LIN {X 0,Y 466.618,Z 479.703,A -85,B 0,C 180,E1 -7650.864,E2 -7650.864} C_VEL
LIN {X 0,Y 466.661,Z 478.907,A -85,B 0,C 180,E1 -7651.727,E2 -7651.727} C_VEL
LIN {X 0,Y 466.686,Z 477.632,A -85,B 0,C 180,E1 -7652.59,E2 -7652.59} C_VEL
LIN {X 0,Y 466.717,Z 474.683,A -85,B 0,C 180,E1 -7653.887,E2 -7653.887} C_VEL
LIN {X 0,Y 466.72,Z 471.998,A -85,B 0,C 180,E1 -7654.752,E2 -7654.752} C_VEL
LIN {X 0,Y 466.841,Z 466.754,A -85,B 0,C 180,E1 -7656.05,E2 -7656.05} C_VEL
LIN {X 0,Y 467.052,Z 459.848,A -85,B 0,C 180,E1 -7657.35,E2 -7657.35} C_VEL
LIN {X 0,Y 467.254,Z 452.312,A -85,B 0,C 180,E1 -7658.434,E2 -7658.434} C_VEL
LIN {X 0,Y 467.532,Z 444.89,A -85,B 0,C 180,E1 -7659.301,E2 -7659.301} C_VEL
LIN {X 0,Y 467.855,Z 436.955,A -85,B 0,C 180,E1 -7660.058,E2 -7660.058} C_VEL
LIN {X 0,Y 468.228,Z 427.08,A -85,B 0,C 180,E1 -7660.815,E2 -7660.815} C_VEL
LIN {X 0,Y 468.601,Z 415.545,A -85,B 0,C 180,E1 -7661.464,E2 -7661.464} C_VEL
LIN {X 0,Y 467.661,Z 405.502,A -85,B 0,C 180,E1 -7661.898,E2 -7661.898} C_VEL
LIN {X 0,Y 466.839,Z 397.843,A -85,B 0,C 180,E1 -7662.168,E2 -7662.168} C_VEL
LIN {X 0,Y 467.003,Z 388.045,A -85,B 0,C 180,E1 -7665.603,E2 -7665.603} C_VEL
LIN {X 0,Y 467.199,Z 379.627,A -85,B 0,C 180,E1 -7668.612,E2 -7668.612} C_VEL
LIN {X 0,Y 467.394,Z 371.372,A -85,B 0,C 180,E1 -7671.617,E2 -7671.617} C_VEL
LIN {X 0,Y 467.717,Z 362.707,A -85,B 0,C 180,E1 -7674.882,E2 -7674.882} C_VEL
LIN {X 0,Y 468.042,Z 355.361,A -85,B 0,C 180,E1 -7677.743,E2 -7677.743} C_VEL
LIN {X 0,Y 468.487,Z 348.104,A -85,B 0,C 180,E1 -7680.668,E2 -7680.668} C_VEL
LIN {X 0,Y 468.775,Z 342.812,A -85,B 0,C 180,E1 -7682.905,E2 -7682.905} C_VEL
LIN {X 0,Y 468.213,Z 338.68,A -85,B 0,C 180,E1 -7684.778,E2 -7684.778} C_VEL
LIN {X 0,Y 467.554,Z 335.06,A -85,B 0,C 180,E1 -7686.558,E2 -7686.558} C_VEL
LIN {X 0,Y 467.588,Z 335.057,A -85,B 0,C 180,E1 -7689.145,E2 -7689.145} C_VEL
LIN {X 0,Y 467.593,Z 335.059,A -85,B 0,C 180,E1 -7692.567,E2 -7692.567} C_VEL
LIN {X 0,Y 467.572,Z 335.061,A -85,B 0,C 180,E1 -7695.053,E2 -7695.053} C_VEL
LIN {X 0,Y 467.596,Z 335.055,A -85,B 0,C 180,E1 -7697.44,E2 -7697.44} C_VEL
LIN {X 0,Y 467.565,Z 335.058,A -85,B 0,C 180,E1 -7700.853,E2 -7700.853} C_VEL
LIN {X 0,Y 467.566,Z 335.057,A -85,B 0,C 180,E1 -7704.261,E2 -7704.261} C_VEL
LIN {X 0,Y 467.586,Z 335.055,A -85,B 0,C 180,E1 -7707.321,E2 -7707.321} C_VEL
LIN {X 0,Y 467.575,Z 335.057,A -85,B 0,C 180,E1 -7710.668,E2 -7710.668} C_VEL
LIN {X 0,Y 467.622,Z 335.051,A -85,B 0,C 180,E1 -7713.199,E2 -7713.199} C_VEL
LIN {X 0,Y 467.6,Z 335.055,A -85,B 0,C 180,E1 -7716.468,E2 -7716.468} C_VEL
LIN {X 0,Y 467.629,Z 335.05,A -85,B 0,C 180,E1 -7719.777,E2 -7719.777} C_VEL
LIN {X 0,Y 467.604,Z 335.053,A -85,B 0,C 180,E1 -7722.506,E2 -7722.506} C_VEL
LIN {X 0,Y 467.612,Z 335.051,A -85,B 0,C 180,E1 -7725.196,E2 -7725.196} C_VEL
LIN {X 0,Y 467.663,Z 335.044,A -85,B 0,C 180,E1 -7727.854,E2 -7727.854} C_VEL
LIN {X 0,Y 467.675,Z 335.043,A -85,B 0,C 180,E1 -7731.356,E2 -7731.356} C_VEL
LIN {X 0,Y 467.727,Z 335.037,A -85,B 0,C 180,E1 -7733.962,E2 -7733.962} C_VEL
LIN {X 0,Y 467.856,Z 335.021,A -85,B 0,C 180,E1 -7737.416,E2 -7737.416} C_VEL
LIN {X 0,Y 467.887,Z 335.019,A -85,B 0,C 180,E1 -7739.999,E2 -7739.999} C_VEL
LIN {X 0,Y 467.862,Z 335.021,A -85,B 0,C 180,E1 -7742.582,E2 -7742.582} C_VEL
LIN {X 0,Y 467.741,Z 335.037,A -85,B 0,C 180,E1 -7746.036,E2 -7746.036} C_VEL
LIN {X 0,Y 467.673,Z 335.044,A -85,B 0,C 180,E1 -7748.642,E2 -7748.642} C_VEL
LIN {X 0,Y 467.66,Z 335.047,A -85,B 0,C 180,E1 -7752.144,E2 -7752.144} C_VEL
LIN {X 0,Y 467.642,Z 335.051,A -85,B 0,C 180,E1 -7755.694,E2 -7755.694} C_VEL
LIN {X 0,Y 467.417,Z 335.078,A -85,B 0,C 180,E1 -7758.69,E2 -7758.69} C_VEL
LIN {X 0,Y 467.29,Z 335.094,A -85,B 0,C 180,E1 -7759.321,E2 -7759.321} C_VEL
LIN {X 0,Y 467.198,Z 337.07,A -85,B 0,C 180,E1 -7761.162,E2 -7761.162} C_VEL
LIN {X 0,Y 467.108,Z 340.504,A -85,B 0,C 180,E1 -7763.967,E2 -7763.967} C_VEL
LIN {X 0,Y 466.981,Z 344.105,A -85,B 0,C 180,E1 -7766.838,E2 -7766.838} C_VEL
LIN {X 0,Y 466.91,Z 347.81,A -85,B 0,C 180,E1 -7769.782,E2 -7769.782} C_VEL
LIN {X 0,Y 466.826,Z 351.71,A -85,B 0,C 180,E1 -7772.817,E2 -7772.817} C_VEL
LIN {X 0,Y 466.752,Z 355.321,A -85,B 0,C 180,E1 -7775.6,E2 -7775.6} C_VEL
LIN {X 0,Y 466.727,Z 358.475,A -85,B 0,C 180,E1 -7777.969,E2 -7777.969} C_VEL
LIN {X 0,Y 468.58,Z 368.176,A -85,B 0,C 180,E1 -7778.367,E2 -7778.367} C_VEL
LIN {X 0,Y 468.903,Z 373.407,A -85,B 0,C 180,E1 -7778.617,E2 -7778.617} C_VEL
LIN {X 0,Y 468.593,Z 383.394,A -85,B 0,C 180,E1 -7779.181,E2 -7779.181} C_VEL
LIN {X 0,Y 468.295,Z 392.105,A -85,B 0,C 180,E1 -7779.829,E2 -7779.829} C_VEL
LIN {X 0,Y 467.971,Z 400.816,A -85,B 0,C 180,E1 -7780.646,E2 -7780.646} C_VEL
LIN {X 0,Y 467.701,Z 407.331,A -85,B 0,C 180,E1 -7781.388,E2 -7781.388} C_VEL
LIN {X 0,Y 467.497,Z 413.587,A -85,B 0,C 180,E1 -7782.246,E2 -7782.246} C_VEL
LIN {X 0,Y 467.25,Z 419.139,A -85,B 0,C 180,E1 -7783.167,E2 -7783.167} C_VEL
LIN {X 0,Y 467.064,Z 423.734,A -85,B 0,C 180,E1 -7784.093,E2 -7784.093} C_VEL
LIN {X 0,Y 466.925,Z 427.508,A -85,B 0,C 180,E1 -7785.024,E2 -7785.024} C_VEL
LIN {X 0,Y 466.805,Z 431.088,A -85,B 0,C 180,E1 -7786.166,E2 -7786.166} C_VEL
LIN {X 0,Y 466.685,Z 433.719,A -85,B 0,C 180,E1 -7787.337,E2 -7787.337} C_VEL
LIN {X 0,Y 466.627,Z 435.754,A -85,B 0,C 180,E1 -7788.854,E2 -7788.854} C_VEL
LIN {X 0,Y 466.569,Z 436.187,A -85,B 0,C 180,E1 -7790.192,E2 -7790.192} C_VEL
LIN {X 0,Y 466.6,Z 435.02,A -85,B 0,C 180,E1 -7791.862,E2 -7791.862} C_VEL
LIN {X 0,Y 466.741,Z 432.093,A -85,B 0,C 180,E1 -7793.502,E2 -7793.502} C_VEL
LIN {X 0,Y 466.851,Z 428.469,A -85,B 0,C 180,E1 -7794.747,E2 -7794.747} C_VEL
LIN {X 0,Y 467.024,Z 424.162,A -85,B 0,C 180,E1 -7795.857,E2 -7795.857} C_VEL
LIN {X 0,Y 467.161,Z 420.161,A -85,B 0,C 180,E1 -7796.693,E2 -7796.693} C_VEL
LIN {X 0,Y 467.405,Z 414.019,A -85,B 0,C 180,E1 -7797.737,E2 -7797.737} C_VEL
LIN {X 0,Y 467.69,Z 407.605,A -85,B 0,C 180,E1 -7798.625,E2 -7798.625} C_VEL
LIN {X 0,Y 467.927,Z 399.54,A -85,B 0,C 180,E1 -7799.541,E2 -7799.541} C_VEL
LIN {X 0,Y 468.297,Z 389.393,A -85,B 0,C 180,E1 -7800.442,E2 -7800.442} C_VEL
LIN {X 0,Y 468.624,Z 380.078,A -85,B 0,C 180,E1 -7801.075,E2 -7801.075} C_VEL
LIN {X 0,Y 468.822,Z 371.827,A -85,B 0,C 180,E1 -7801.516,E2 -7801.516} C_VEL
LIN {X 0,Y 468.245,Z 366.243,A -85,B 0,C 180,E1 -7801.783,E2 -7801.783} C_VEL
LIN {X 0,Y 466.751,Z 357.961,A -85,B 0,C 180,E1 -7802.113,E2 -7802.113} C_VEL
LIN {X 0,Y 466.785,Z 354.038,A -85,B 0,C 180,E1 -7805.033,E2 -7805.033} C_VEL
LIN {X 0,Y 466.109,Z 353.155,A -85,B 0,C 180,E1 -7805.745,E2 -7805.745} C_VEL
LIN {X 0,Y 463.245,Z 351.852,A -85,B 0,C 180,E1 -7806.904,E2 -7806.904} C_VEL
LIN {X 0,Y 460.832,Z 350.827,A -85,B 0,C 180,E1 -7807.84,E2 -7807.84} C_VEL
LIN {X 0,Y 459.803,Z 349.971,A -85,B 0,C 180,E1 -7808.561,E2 -7808.561} C_VEL
LIN {X 0,Y 459.721,Z 349.657,A -85,B 0,C 180,E1 -7808.805,E2 -7808.805} C_VEL
LIN {X 0,Y 459.833,Z 346.343,A -85,B 0,C 180,E1 -7811.364,E2 -7811.364} C_VEL
LIN {X 0,Y 459.94,Z 342.592,A -85,B 0,C 180,E1 -7814.287,E2 -7814.287} C_VEL
LIN {X 0,Y 460.076,Z 338.085,A -85,B 0,C 180,E1 -7817.855,E2 -7817.855} C_VEL
LIN {X 0,Y 460.088,Z 336.115,A -85,B 0,C 180,E1 -7819.437,E2 -7819.437} C_VEL
LIN {X 0,Y 460.626,Z 335.921,A -85,B 0,C 180,E1 -7822.618,E2 -7822.618} C_VEL
LIN {X 0,Y 460.685,Z 335.914,A -85,B 0,C 180,E1 -7824.747,E2 -7824.747} C_VEL
LIN {X 0,Y 460.815,Z 335.897,A -85,B 0,C 180,E1 -7827.376,E2 -7827.376} C_VEL
LIN {X 0,Y 460.842,Z 335.895,A -85,B 0,C 180,E1 -7829.999,E2 -7829.999} C_VEL
LIN {X 0,Y 460.816,Z 335.897,A -85,B 0,C 180,E1 -7832.621,E2 -7832.621} C_VEL
LIN {X 0,Y 460.706,Z 335.912,A -85,B 0,C 180,E1 -7836.129,E2 -7836.129} C_VEL
LIN {X 0,Y 460.618,Z 335.921,A -85,B 0,C 180,E1 -7838.775,E2 -7838.775} C_VEL
LIN {X 0,Y 460.621,Z 335.921,A -85,B 0,C 180,E1 -7842.456,E2 -7842.456} C_VEL
LIN {X 0,Y 460.587,Z 335.926,A -85,B 0,C 180,E1 -7845.997,E2 -7845.997} C_VEL
LIN {X 0,Y 460.558,Z 335.929,A -85,B 0,C 180,E1 -7848.901,E2 -7848.901} C_VEL
LIN {X 0,Y 460.502,Z 335.939,A -85,B 0,C 180,E1 -7851.485,E2 -7851.485} C_VEL
LIN {X 0,Y 460.529,Z 335.931,A -85,B 0,C 180,E1 -7854.332,E2 -7854.332} C_VEL
LIN {X 0,Y 460.57,Z 335.929,A -85,B 0,C 180,E1 -7857.242,E2 -7857.242} C_VEL
LIN {X 0,Y 460.513,Z 335.934,A -85,B 0,C 180,E1 -7860.238,E2 -7860.238} C_VEL
LIN {X 0,Y 460.515,Z 335.936,A -85,B 0,C 180,E1 -7863.324,E2 -7863.324} C_VEL
LIN {X 0,Y 460.466,Z 335.941,A -85,B 0,C 180,E1 -7866.529,E2 -7866.529} C_VEL
LIN {X 0,Y 460.564,Z 335.928,A -85,B 0,C 180,E1 -7869.857,E2 -7869.857} C_VEL
LIN {X 0,Y 460.527,Z 335.934,A -85,B 0,C 180,E1 -7872.904,E2 -7872.904} C_VEL
LIN {X 0,Y 460.508,Z 335.935,A -85,B 0,C 180,E1 -7875.829,E2 -7875.829} C_VEL
LIN {X 0,Y 460.528,Z 335.934,A -85,B 0,C 180,E1 -7878.99,E2 -7878.99} C_VEL
LIN {X 0,Y 460.533,Z 335.933,A -85,B 0,C 180,E1 -7881.269,E2 -7881.269} C_VEL
LIN {X 0,Y 460.499,Z 335.938,A -85,B 0,C 180,E1 -7884.555,E2 -7884.555} C_VEL
LIN {X 0,Y 460.518,Z 335.934,A -85,B 0,C 180,E1 -7887.716,E2 -7887.716} C_VEL
LIN {X 0,Y 460.533,Z 335.933,A -85,B 0,C 180,E1 -7890.77,E2 -7890.77} C_VEL
LIN {X 0,Y 460.549,Z 335.93,A -85,B 0,C 180,E1 -7893.735,E2 -7893.735} C_VEL
LIN {X 0,Y 460.534,Z 335.934,A -85,B 0,C 180,E1 -7896.625,E2 -7896.625} C_VEL
LIN {X 0,Y 460.559,Z 335.927,A -85,B 0,C 180,E1 -7899.454,E2 -7899.454} C_VEL
LIN {X 0,Y 460.546,Z 335.932,A -85,B 0,C 180,E1 -7902.231,E2 -7902.231} C_VEL
LIN {X 0,Y 460.556,Z 335.929,A -85,B 0,C 180,E1 -7904.966,E2 -7904.966} C_VEL
LIN {X 0,Y 460.616,Z 335.923,A -85,B 0,C 180,E1 -7907.667,E2 -7907.667} C_VEL
LIN {X 0,Y 460.617,Z 335.922,A -85,B 0,C 180,E1 -7911.225,E2 -7911.225} C_VEL
LIN {X 0,Y 460.699,Z 335.913,A -85,B 0,C 180,E1 -7913.871,E2 -7913.871} C_VEL
LIN {X 0,Y 460.815,Z 335.898,A -85,B 0,C 180,E1 -7917.378,E2 -7917.378} C_VEL
LIN {X 0,Y 460.841,Z 335.895,A -85,B 0,C 180,E1 -7920.001,E2 -7920.001} C_VEL
LIN {X 0,Y 460.816,Z 335.897,A -85,B 0,C 180,E1 -7922.623,E2 -7922.623} C_VEL
LIN {X 0,Y 460.699,Z 335.912,A -85,B 0,C 180,E1 -7926.131,E2 -7926.131} C_VEL
LIN {X 0,Y 460.619,Z 335.921,A -85,B 0,C 180,E1 -7928.777,E2 -7928.777} C_VEL
LIN {X 0,Y 460.624,Z 335.921,A -85,B 0,C 180,E1 -7932.458,E2 -7932.458} C_VEL
LIN {X 0,Y 460.59,Z 335.926,A -85,B 0,C 180,E1 -7935.999,E2 -7935.999} C_VEL
LIN {X 0,Y 460.561,Z 335.929,A -85,B 0,C 180,E1 -7938.903,E2 -7938.903} C_VEL
LIN {X 0,Y 460.507,Z 335.937,A -85,B 0,C 180,E1 -7941.487,E2 -7941.487} C_VEL
LIN {X 0,Y 460.534,Z 335.93,A -85,B 0,C 180,E1 -7944.333,E2 -7944.333} C_VEL
LIN {X 0,Y 460.576,Z 335.929,A -85,B 0,C 180,E1 -7947.244,E2 -7947.244} C_VEL
LIN {X 0,Y 460.519,Z 335.933,A -85,B 0,C 180,E1 -7950.24,E2 -7950.24} C_VEL
LIN {X 0,Y 460.522,Z 335.936,A -85,B 0,C 180,E1 -7953.326,E2 -7953.326} C_VEL
LIN {X 0,Y 460.472,Z 335.94,A -85,B 0,C 180,E1 -7956.53,E2 -7956.53} C_VEL
LIN {X 0,Y 460.538,Z 335.933,A -85,B 0,C 180,E1 -7958.899,E2 -7958.899} C_VEL
LIN {X 0,Y 460.517,Z 335.935,A -85,B 0,C 180,E1 -7962.183,E2 -7962.183} C_VEL
LIN {X 0,Y 460.514,Z 335.936,A -85,B 0,C 180,E1 -7965.413,E2 -7965.413} C_VEL
LIN {X 0,Y 460.53,Z 335.934,A -85,B 0,C 180,E1 -7968.398,E2 -7968.398} C_VEL
LIN {X 0,Y 460.522,Z 335.934,A -85,B 0,C 180,E1 -7971.268,E2 -7971.268} C_VEL
LIN {X 0,Y 460.543,Z 336.026,A -85,B 0,C 180,E1 -7973.553,E2 -7973.553} C_VEL
LIN {X 0,Y 461.613,Z 341.991,A -85,B 0,C 180,E1 -7976.242,E2 -7976.242} C_VEL
LIN {X 0,Y 461.711,Z 345.667,A -85,B 0,C 180,E1 -7977.81,E2 -7977.81} C_VEL
LIN {X 0,Y 461.273,Z 353.052,A -85,B 0,C 180,E1 -7980.822,E2 -7980.822} C_VEL
LIN {X 0,Y 460.829,Z 361.444,A -85,B 0,C 180,E1 -7984.132,E2 -7984.132} C_VEL
LIN {X 0,Y 460.494,Z 369.168,A -85,B 0,C 180,E1 -7987.098,E2 -7987.098} C_VEL
LIN {X 0,Y 460.207,Z 377.901,A -85,B 0,C 180,E1 -7990.37,E2 -7990.37} C_VEL
LIN {X 0,Y 460.009,Z 386.643,A -85,B 0,C 180,E1 -7993.583,E2 -7993.583} C_VEL
LIN {X 0,Y 459.783,Z 395.418,A -85,B 0,C 180,E1 -7996.746,E2 -7996.746} C_VEL
LIN {X 0,Y 459.781,Z 398.053,A -85,B 0,C 180,E1 -7997.693,E2 -7997.693} C_VEL
LIN {X 0,Y 461,Z 410.041,A -85,B 0,C 180,E1 -7998.11,E2 -7998.11} C_VEL
LIN {X 0,Y 461.555,Z 417.186,A -85,B 0,C 180,E1 -7998.453,E2 -7998.453} C_VEL
LIN {X 0,Y 461.209,Z 428.346,A -85,B 0,C 180,E1 -7999.132,E2 -7999.132} C_VEL
LIN {X 0,Y 460.876,Z 436.733,A -85,B 0,C 180,E1 -7999.79,E2 -7999.79} C_VEL
LIN {X 0,Y 460.533,Z 444.67,A -85,B 0,C 180,E1 -8000.559,E2 -8000.559} C_VEL
LIN {X 0,Y 460.247,Z 452.093,A -85,B 0,C 180,E1 -8001.439,E2 -8001.439} C_VEL
LIN {X 0,Y 459.972,Z 459.627,A -85,B 0,C 180,E1 -8002.539,E2 -8002.539} C_VEL
LIN {X 0,Y 459.749,Z 466.524,A -85,B 0,C 180,E1 -8003.858,E2 -8003.858} C_VEL
LIN {X 0,Y 459.651,Z 471.744,A -85,B 0,C 180,E1 -8005.177,E2 -8005.177} C_VEL
LIN {X 0,Y 459.611,Z 474.418,A -85,B 0,C 180,E1 -8006.056,E2 -8006.056} C_VEL
LIN {X 0,Y 459.609,Z 477.345,A -85,B 0,C 180,E1 -8007.372,E2 -8007.372} C_VEL
LIN {X 0,Y 459.57,Z 478.608,A -85,B 0,C 180,E1 -8008.248,E2 -8008.248} C_VEL
LIN {X 0,Y 459.551,Z 479.391,A -85,B 0,C 180,E1 -8009.125,E2 -8009.125} C_VEL
LIN {X 0,Y 459.531,Z 479.678,A -85,B 0,C 180,E1 -8010.001,E2 -8010.001} C_VEL
LIN {X 0,Y 459.551,Z 479.371,A -85,B 0,C 180,E1 -8010.877,E2 -8010.877} C_VEL
LIN {X 0,Y 459.57,Z 478.576,A -85,B 0,C 180,E1 -8011.754,E2 -8011.754} C_VEL
LIN {X 0,Y 459.609,Z 477.301,A -85,B 0,C 180,E1 -8012.63,E2 -8012.63} C_VEL
LIN {X 0,Y 459.61,Z 474.35,A -85,B 0,C 180,E1 -8013.947,E2 -8013.947} C_VEL
LIN {X 0,Y 459.651,Z 471.666,A -85,B 0,C 180,E1 -8014.825,E2 -8014.825} C_VEL
LIN {X 0,Y 459.75,Z 466.419,A -85,B 0,C 180,E1 -8016.144,E2 -8016.144} C_VEL
LIN {X 0,Y 459.978,Z 459.518,A -85,B 0,C 180,E1 -8017.463,E2 -8017.463} C_VEL
LIN {X 0,Y 460.218,Z 451.988,A -85,B 0,C 180,E1 -8018.564,E2 -8018.564} C_VEL
LIN {X 0,Y 460.521,Z 444.576,A -85,B 0,C 180,E1 -8019.443,E2 -8019.443} C_VEL
LIN {X 0,Y 460.861,Z 436.653,A -85,B 0,C 180,E1 -8020.212,E2 -8020.212} C_VEL
LIN {X 0,Y 461.176,Z 428.297,A -85,B 0,C 180,E1 -8020.871,E2 -8020.871} C_VEL
LIN {X 0,Y 461.598,Z 417.276,A -85,B 0,C 180,E1 -8021.548,E2 -8021.548} C_VEL
LIN {X 0,Y 460.674,Z 405.859,A -85,B 0,C 180,E1 -8022.064,E2 -8022.064} C_VEL
LIN {X 0,Y 459.735,Z 397.524,A -85,B 0,C 180,E1 -8022.359,E2 -8022.359} C_VEL
LIN {X 0,Y 459.939,Z 388.146,A -85,B 0,C 180,E1 -8025.707,E2 -8025.707} C_VEL
LIN {X 0,Y 460.145,Z 378.789,A -85,B 0,C 180,E1 -8029.125,E2 -8029.125} C_VEL
LIN {X 0,Y 460.356,Z 371.132,A -85,B 0,C 180,E1 -8031.965,E2 -8031.965} C_VEL
LIN {X 0,Y 460.729,Z 362.485,A -85,B 0,C 180,E1 -8035.286,E2 -8035.286} C_VEL
LIN {X 0,Y 461.146,Z 354.024,A -85,B 0,C 180,E1 -8038.691,E2 -8038.691} C_VEL
LIN {X 0,Y 461.544,Z 348.034,A -85,B 0,C 180,E1 -8041.181,E2 -8041.181} C_VEL
LIN {X 0,Y 461.713,Z 343.331,A -85,B 0,C 180,E1 -8043.229,E2 -8043.229} C_VEL
LIN {X 0,Y 461.004,Z 338.695,A -85,B 0,C 180,E1 -8045.403,E2 -8045.403} C_VEL
LIN {X 0,Y 460.519,Z 335.936,A -85,B 0,C 180,E1 -8046.799,E2 -8046.799} C_VEL
LIN {X 0,Y 460.538,Z 335.937,A -85,B 0,C 180,E1 -8049.863,E2 -8049.863} C_VEL
LIN {X 0,Y 460.519,Z 335.941,A -85,B 0,C 180,E1 -8052.901,E2 -8052.901} C_VEL
LIN {X 0,Y 460.513,Z 335.938,A -85,B 0,C 180,E1 -8055.831,E2 -8055.831} C_VEL
LIN {X 0,Y 460.537,Z 335.934,A -85,B 0,C 180,E1 -8058.989,E2 -8058.989} C_VEL
LIN {X 0,Y 460.524,Z 335.936,A -85,B 0,C 180,E1 -8061.266,E2 -8061.266} C_VEL
LIN {X 0,Y 460.515,Z 335.937,A -85,B 0,C 180,E1 -8064.554,E2 -8064.554} C_VEL
LIN {X 0,Y 460.536,Z 335.932,A -85,B 0,C 180,E1 -8067.715,E2 -8067.715} C_VEL
LIN {X 0,Y 460.545,Z 335.932,A -85,B 0,C 180,E1 -8070.769,E2 -8070.769} C_VEL
LIN {X 0,Y 460.566,Z 335.929,A -85,B 0,C 180,E1 -8073.734,E2 -8073.734} C_VEL
LIN {X 0,Y 460.553,Z 335.931,A -85,B 0,C 180,E1 -8076.624,E2 -8076.624} C_VEL
LIN {X 0,Y 460.557,Z 335.929,A -85,B 0,C 180,E1 -8079.452,E2 -8079.452} C_VEL
LIN {X 0,Y 460.556,Z 335.931,A -85,B 0,C 180,E1 -8082.229,E2 -8082.229} C_VEL
LIN {X 0,Y 460.571,Z 335.929,A -85,B 0,C 180,E1 -8084.964,E2 -8084.964} C_VEL
LIN {X 0,Y 460.616,Z 335.923,A -85,B 0,C 180,E1 -8088.559,E2 -8088.559} C_VEL
LIN {X 0,Y 460.625,Z 335.921,A -85,B 0,C 180,E1 -8091.223,E2 -8091.223} C_VEL
LIN {X 0,Y 460.691,Z 335.913,A -85,B 0,C 180,E1 -8093.869,E2 -8093.869} C_VEL
LIN {X 0,Y 460.796,Z 335.901,A -85,B 0,C 180,E1 -8097.377,E2 -8097.377} C_VEL
LIN {X 0,Y 460.857,Z 335.895,A -85,B 0,C 180,E1 -8099.999,E2 -8099.999} C_VEL
LIN {X 0,Y 460.803,Z 335.9,A -85,B 0,C 180,E1 -8102.622,E2 -8102.622} C_VEL
LIN {X 0,Y 460.706,Z 335.913,A -85,B 0,C 180,E1 -8106.129,E2 -8106.129} C_VEL
LIN {X 0,Y 460.623,Z 335.922,A -85,B 0,C 180,E1 -8108.775,E2 -8108.775} C_VEL
LIN {X 0,Y 460.618,Z 335.923,A -85,B 0,C 180,E1 -8112.444,E2 -8112.444} C_VEL
LIN {X 0,Y 460.581,Z 335.93,A -85,B 0,C 180,E1 -8115.987,E2 -8115.987} C_VEL
LIN {X 0,Y 460.34,Z 335.959,A -85,B 0,C 180,E1 -8118.815,E2 -8118.815} C_VEL
LIN {X 0,Y 460.194,Z 336.061,A -85,B 0,C 180,E1 -8119.631,E2 -8119.631} C_VEL
LIN {X 0,Y 460.092,Z 339.461,A -85,B 0,C 180,E1 -8122.449,E2 -8122.449} C_VEL
LIN {X 0,Y 459.98,Z 343.335,A -85,B 0,C 180,E1 -8125.648,E2 -8125.648} C_VEL
LIN {X 0,Y 459.906,Z 346.641,A -85,B 0,C 180,E1 -8128.275,E2 -8128.275} C_VEL
LIN {X 0,Y 459.818,Z 350.456,A -85,B 0,C 180,E1 -8131.308,E2 -8131.308} C_VEL
LIN {X 0,Y 459.724,Z 354.451,A -85,B 0,C 180,E1 -8134.445,E2 -8134.445} C_VEL
LIN {X 0,Y 459.655,Z 358.766,A -85,B 0,C 180,E1 -8137.772,E2 -8137.772} C_VEL
LIN {X 0,Y 461.793,Z 370.032,A -85,B 0,C 180,E1 -8138.258,E2 -8138.258} C_VEL
LIN {X 0,Y 461.881,Z 376.837,A -85,B 0,C 180,E1 -8138.597,E2 -8138.597} C_VEL
LIN {X 0,Y 461.585,Z 385.85,A -85,B 0,C 180,E1 -8139.163,E2 -8139.163} C_VEL
LIN {X 0,Y 461.26,Z 393.763,A -85,B 0,C 180,E1 -8139.785,E2 -8139.785} C_VEL
LIN {X 0,Y 461.016,Z 400.657,A -85,B 0,C 180,E1 -8140.443,E2 -8140.443} C_VEL
LIN {X 0,Y 460.682,Z 408.035,A -85,B 0,C 180,E1 -8141.297,E2 -8141.297} C_VEL
LIN {X 0,Y 460.464,Z 414.342,A -85,B 0,C 180,E1 -8142.186,E2 -8142.186} C_VEL
LIN {X 0,Y 460.11,Z 421.406,A -85,B 0,C 180,E1 -8143.419,E2 -8143.419} C_VEL
LIN {X 0,Y 459.929,Z 426.867,A -85,B 0,C 180,E1 -8144.659,E2 -8144.659} C_VEL
LIN {X 0,Y 459.763,Z 430.963,A -85,B 0,C 180,E1 -8145.925,E2 -8145.925} C_VEL
LIN {X 0,Y 459.611,Z 433.924,A -85,B 0,C 180,E1 -8147.219,E2 -8147.219} C_VEL
LIN {X 0,Y 459.543,Z 435.772,A -85,B 0,C 180,E1 -8148.535,E2 -8148.535} C_VEL
LIN {X 0,Y 459.496,Z 436.55,A -85,B 0,C 180,E1 -8150.029,E2 -8150.029} C_VEL
LIN {X 0,Y 459.485,Z 436.038,A -85,B 0,C 180,E1 -8151.264,E2 -8151.264} C_VEL
LIN {X 0,Y 459.558,Z 434.181,A -85,B 0,C 180,E1 -8152.675,E2 -8152.675} C_VEL
LIN {X 0,Y 459.646,Z 432.817,A -85,B 0,C 180,E1 -8153.393,E2 -8153.393} C_VEL
LIN {X 0,Y 459.757,Z 429.915,A -85,B 0,C 180,E1 -8154.487,E2 -8154.487} C_VEL
LIN {X 0,Y 459.968,Z 424.797,A -85,B 0,C 180,E1 -8155.869,E2 -8155.869} C_VEL
LIN {X 0,Y 460.153,Z 419.781,A -85,B 0,C 180,E1 -8156.921,E2 -8156.921} C_VEL
LIN {X 0,Y 460.326,Z 415.314,A -85,B 0,C 180,E1 -8157.698,E2 -8157.698} C_VEL
LIN {X 0,Y 460.584,Z 409.931,A -85,B 0,C 180,E1 -8158.492,E2 -8158.492} C_VEL
LIN {X 0,Y 460.871,Z 402.393,A -85,B 0,C 180,E1 -8159.405,E2 -8159.405} C_VEL
LIN {X 0,Y 461.116,Z 395.587,A -85,B 0,C 180,E1 -8160.088,E2 -8160.088} C_VEL
LIN {X 0,Y 461.409,Z 387.767,A -85,B 0,C 180,E1 -8160.736,E2 -8160.736} C_VEL
LIN {X 0,Y 461.704,Z 379.555,A -85,B 0,C 180,E1 -8161.285,E2 -8161.285} C_VEL
LIN {X 0,Y 461.898,Z 371.097,A -85,B 0,C 180,E1 -8161.732,E2 -8161.732} C_VEL
LIN {X 0,Y 460.131,Z 360.919,A -85,B 0,C 180,E1 -8162.182,E2 -8162.182} C_VEL
LIN {X 0,Y 459.686,Z 358.242,A -85,B 0,C 180,E1 -8162.308,E2 -8162.308} C_VEL
LIN {X 0,Y 459.695,Z 354.608,A -85,B 0,C 180,E1 -8165.037,E2 -8165.037} C_VEL
LIN {X 0,Y 459.708,Z 351.33,A -85,B 0,C 180,E1 -8167.529,E2 -8167.529} C_VEL
LIN {X 0,Y 459.721,Z 349.657,A -85,B 0,C 180,E1 -8168.805,E2 -8168.805} C_VEL
LIN {X 0,Y 459.063,Z 348.78,A -85,B 0,C 180,E1 -8169.528,E2 -8169.528} C_VEL
LIN {X 0,Y 456.226,Z 347.51,A -85,B 0,C 180,E1 -8170.708,E2 -8170.708} C_VEL
LIN {X 0,Y 453.841,Z 346.514,A -85,B 0,C 180,E1 -8171.66,E2 -8171.66} C_VEL
LIN {X 0,Y 452.842,Z 345.676,A -85,B 0,C 180,E1 -8172.394,E2 -8172.394} C_VEL
LIN {X 0,Y 452.774,Z 345.363,A -85,B 0,C 180,E1 -8172.642,E2 -8172.642} C_VEL
LIN {X 0,Y 452.851,Z 341.597,A -85,B 0,C 180,E1 -8175.621,E2 -8175.621} C_VEL
LIN {X 0,Y 453.018,Z 338.172,A -85,B 0,C 180,E1 -8178.364,E2 -8178.364} C_VEL
LIN {X 0,Y 453.027,Z 337.053,A -85,B 0,C 180,E1 -8179.27,E2 -8179.27} C_VEL
LIN {X 0,Y 453.577,Z 336.8,A -85,B 0,C 180,E1 -8182.581,E2 -8182.581} C_VEL
LIN {X 0,Y 453.657,Z 336.79,A -85,B 0,C 180,E1 -8184.665,E2 -8184.665} C_VEL
LIN {X 0,Y 453.755,Z 336.776,A -85,B 0,C 180,E1 -8187.336,E2 -8187.336} C_VEL
LIN {X 0,Y 453.812,Z 336.771,A -85,B 0,C 180,E1 -8189.999,E2 -8189.999} C_VEL
LIN {X 0,Y 453.756,Z 336.776,A -85,B 0,C 180,E1 -8192.662,E2 -8192.662} C_VEL
LIN {X 0,Y 453.672,Z 336.788,A -85,B 0,C 180,E1 -8196.224,E2 -8196.224} C_VEL
LIN {X 0,Y 453.582,Z 336.797,A -85,B 0,C 180,E1 -8198.912,E2 -8198.912} C_VEL
LIN {X 0,Y 453.589,Z 336.798,A -85,B 0,C 180,E1 -8202.55,E2 -8202.55} C_VEL
LIN {X 0,Y 453.531,Z 336.806,A -85,B 0,C 180,E1 -8206.195,E2 -8206.195} C_VEL
LIN {X 0,Y 453.507,Z 336.808,A -85,B 0,C 180,E1 -8209.04,E2 -8209.04} C_VEL
LIN {X 0,Y 453.463,Z 336.814,A -85,B 0,C 180,E1 -8211.835,E2 -8211.835} C_VEL
LIN {X 0,Y 453.5,Z 336.807,A -85,B 0,C 180,E1 -8214.734,E2 -8214.734} C_VEL
LIN {X 0,Y 453.524,Z 336.805,A -85,B 0,C 180,E1 -8217.961,E2 -8217.961} C_VEL
LIN {X 0,Y 453.469,Z 336.811,A -85,B 0,C 180,E1 -8220.758,E2 -8220.758} C_VEL
LIN {X 0,Y 453.463,Z 336.812,A -85,B 0,C 180,E1 -8223.912,E2 -8223.912} C_VEL
LIN {X 0,Y 453.458,Z 336.816,A -85,B 0,C 180,E1 -8227.187,E2 -8227.187} C_VEL
LIN {X 0,Y 453.518,Z 336.808,A -85,B 0,C 180,E1 -8229.445,E2 -8229.445} C_VEL
LIN {X 0,Y 453.477,Z 336.812,A -85,B 0,C 180,E1 -8232.991,E2 -8232.991} C_VEL
LIN {X 0,Y 453.462,Z 336.813,A -85,B 0,C 180,E1 -8235.78,E2 -8235.78} C_VEL
LIN {X 0,Y 453.481,Z 336.811,A -85,B 0,C 180,E1 -8238.211,E2 -8238.211} C_VEL
LIN {X 0,Y 453.518,Z 336.808,A -85,B 0,C 180,E1 -8240.787,E2 -8240.787} C_VEL
LIN {X 0,Y 453.443,Z 336.814,A -85,B 0,C 180,E1 -8243.918,E2 -8243.918} C_VEL
LIN {X 0,Y 453.468,Z 336.813,A -85,B 0,C 180,E1 -8247.151,E2 -8247.151} C_VEL
LIN {X 0,Y 453.499,Z 336.809,A -85,B 0,C 180,E1 -8250.271,E2 -8250.271} C_VEL
LIN {X 0,Y 453.495,Z 336.808,A -85,B 0,C 180,E1 -8253.295,E2 -8253.295} C_VEL
LIN {X 0,Y 453.492,Z 336.81,A -85,B 0,C 180,E1 -8256.239,E2 -8256.239} C_VEL
LIN {X 0,Y 453.494,Z 336.808,A -85,B 0,C 180,E1 -8259.119,E2 -8259.119} C_VEL
LIN {X 0,Y 453.499,Z 336.809,A -85,B 0,C 180,E1 -8261.945,E2 -8261.945} C_VEL
LIN {X 0,Y 453.536,Z 336.806,A -85,B 0,C 180,E1 -8264.727,E2 -8264.727} C_VEL
LIN {X 0,Y 453.589,Z 336.797,A -85,B 0,C 180,E1 -8267.473,E2 -8267.473} C_VEL
LIN {X 0,Y 453.581,Z 336.798,A -85,B 0,C 180,E1 -8271.087,E2 -8271.087} C_VEL
LIN {X 0,Y 453.666,Z 336.789,A -85,B 0,C 180,E1 -8273.776,E2 -8273.776} C_VEL
LIN {X 0,Y 453.755,Z 336.777,A -85,B 0,C 180,E1 -8277.338,E2 -8277.338} C_VEL
LIN {X 0,Y 453.811,Z 336.771,A -85,B 0,C 180,E1 -8280.001,E2 -8280.001} C_VEL
LIN {X 0,Y 453.757,Z 336.776,A -85,B 0,C 180,E1 -8282.664,E2 -8282.664} C_VEL
LIN {X 0,Y 453.667,Z 336.788,A -85,B 0,C 180,E1 -8286.226,E2 -8286.226} C_VEL
LIN {X 0,Y 453.583,Z 336.797,A -85,B 0,C 180,E1 -8288.914,E2 -8288.914} C_VEL
LIN {X 0,Y 453.591,Z 336.797,A -85,B 0,C 180,E1 -8292.552,E2 -8292.552} C_VEL
LIN {X 0,Y 453.535,Z 336.805,A -85,B 0,C 180,E1 -8296.197,E2 -8296.197} C_VEL
LIN {X 0,Y 453.511,Z 336.808,A -85,B 0,C 180,E1 -8299.042,E2 -8299.042} C_VEL
LIN {X 0,Y 453.467,Z 336.813,A -85,B 0,C 180,E1 -8301.837,E2 -8301.837} C_VEL
LIN {X 0,Y 453.506,Z 336.807,A -85,B 0,C 180,E1 -8304.736,E2 -8304.736} C_VEL
LIN {X 0,Y 453.531,Z 336.804,A -85,B 0,C 180,E1 -8307.962,E2 -8307.962} C_VEL
LIN {X 0,Y 453.475,Z 336.811,A -85,B 0,C 180,E1 -8310.76,E2 -8310.76} C_VEL
LIN {X 0,Y 453.471,Z 336.811,A -85,B 0,C 180,E1 -8313.914,E2 -8313.914} C_VEL
LIN {X 0,Y 453.464,Z 336.815,A -85,B 0,C 180,E1 -8317.189,E2 -8317.189} C_VEL
LIN {X 0,Y 453.499,Z 336.81,A -85,B 0,C 180,E1 -8319.449,E2 -8319.449} C_VEL
LIN {X 0,Y 453.462,Z 336.815,A -85,B 0,C 180,E1 -8322.996,E2 -8322.996} C_VEL
LIN {X 0,Y 453.467,Z 336.812,A -85,B 0,C 180,E1 -8325.781,E2 -8325.781} C_VEL
LIN {X 0,Y 453.476,Z 336.812,A -85,B 0,C 180,E1 -8328.211,E2 -8328.211} C_VEL
LIN {X 0,Y 453.511,Z 336.807,A -85,B 0,C 180,E1 -8330.791,E2 -8330.791} C_VEL
LIN {X 0,Y 453.517,Z 336.992,A -85,B 0,C 180,E1 -8333.403,E2 -8333.403} C_VEL
LIN {X 0,Y 454.596,Z 343.067,A -85,B 0,C 180,E1 -8336.184,E2 -8336.184} C_VEL
LIN {X 0,Y 454.638,Z 347.832,A -85,B 0,C 180,E1 -8338.236,E2 -8338.236} C_VEL
LIN {X 0,Y 454.156,Z 355.343,A -85,B 0,C 180,E1 -8341.334,E2 -8341.334} C_VEL
LIN {X 0,Y 453.752,Z 362.759,A -85,B 0,C 180,E1 -8344.3,E2 -8344.3} C_VEL
LIN {X 0,Y 453.427,Z 370.183,A -85,B 0,C 180,E1 -8347.203,E2 -8347.203} C_VEL
LIN {X 0,Y 453.122,Z 378.885,A -85,B 0,C 180,E1 -8350.522,E2 -8350.522} C_VEL
LIN {X 0,Y 452.898,Z 387.629,A -85,B 0,C 180,E1 -8353.782,E2 -8353.782} C_VEL
LIN {X 0,Y 452.693,Z 396.338,A -85,B 0,C 180,E1 -8356.992,E2 -8356.992} C_VEL
LIN {X 0,Y 452.707,Z 397.739,A -85,B 0,C 180,E1 -8357.505,E2 -8357.505} C_VEL
LIN {X 0,Y 454.03,Z 410.787,A -85,B 0,C 180,E1 -8357.983,E2 -8357.983} C_VEL
LIN {X 0,Y 454.556,Z 418.104,A -85,B 0,C 180,E1 -8358.348,E2 -8358.348} C_VEL
LIN {X 0,Y 454.22,Z 427.901,A -85,B 0,C 180,E1 -8358.962,E2 -8358.962} C_VEL
LIN {X 0,Y 453.852,Z 436.31,A -85,B 0,C 180,E1 -8359.631,E2 -8359.631} C_VEL
LIN {X 0,Y 453.512,Z 444.265,A -85,B 0,C 180,E1 -8360.412,E2 -8360.412} C_VEL
LIN {X 0,Y 453.204,Z 451.704,A -85,B 0,C 180,E1 -8361.305,E2 -8361.305} C_VEL
LIN {X 0,Y 452.899,Z 459.25,A -85,B 0,C 180,E1 -8362.422,E2 -8362.422} C_VEL
LIN {X 0,Y 452.66,Z 466.165,A -85,B 0,C 180,E1 -8363.762,E2 -8363.762} C_VEL
LIN {X 0,Y 452.582,Z 471.394,A -85,B 0,C 180,E1 -8365.102,E2 -8365.102} C_VEL
LIN {X 0,Y 452.509,Z 474.072,A -85,B 0,C 180,E1 -8365.993,E2 -8365.993} C_VEL
LIN {X 0,Y 452.533,Z 477.005,A -85,B 0,C 180,E1 -8367.331,E2 -8367.331} C_VEL
LIN {X 0,Y 452.483,Z 478.27,A -85,B 0,C 180,E1 -8368.221,E2 -8368.221} C_VEL
LIN {X 0,Y 452.486,Z 479.058,A -85,B 0,C 180,E1 -8369.111,E2 -8369.111} C_VEL
LIN {X 0,Y 452.464,Z 479.346,A -85,B 0,C 180,E1 -8370.001,E2 -8370.001} C_VEL
LIN {X 0,Y 452.486,Z 479.04,A -85,B 0,C 180,E1 -8370.891,E2 -8370.891} C_VEL
LIN {X 0,Y 452.483,Z 478.245,A -85,B 0,C 180,E1 -8371.781,E2 -8371.781} C_VEL
LIN {X 0,Y 452.534,Z 476.974,A -85,B 0,C 180,E1 -8372.672,E2 -8372.672} C_VEL
LIN {X 0,Y 452.508,Z 474.024,A -85,B 0,C 180,E1 -8374.009,E2 -8374.009} C_VEL
LIN {X 0,Y 452.582,Z 471.344,A -85,B 0,C 180,E1 -8374.901,E2 -8374.901} C_VEL
LIN {X 0,Y 452.662,Z 466.101,A -85,B 0,C 180,E1 -8376.24,E2 -8376.24} C_VEL
LIN {X 0,Y 452.903,Z 459.207,A -85,B 0,C 180,E1 -8377.58,E2 -8377.58} C_VEL
LIN {X 0,Y 453.188,Z 451.685,A -85,B 0,C 180,E1 -8378.698,E2 -8378.698} C_VEL
LIN {X 0,Y 453.511,Z 444.28,A -85,B 0,C 180,E1 -8379.591,E2 -8379.591} C_VEL
LIN {X 0,Y 453.848,Z 436.365,A -85,B 0,C 180,E1 -8380.372,E2 -8380.372} C_VEL
LIN {X 0,Y 454.202,Z 428.025,A -85,B 0,C 180,E1 -8381.04,E2 -8381.04} C_VEL
LIN {X 0,Y 454.615,Z 417.333,A -85,B 0,C 180,E1 -8381.713,E2 -8381.713} C_VEL
LIN {X 0,Y 453.637,Z 405.688,A -85,B 0,C 180,E1 -8382.254,E2 -8382.254} C_VEL
LIN {X 0,Y 452.666,Z 397.221,A -85,B 0,C 180,E1 -8382.555,E2 -8382.555} C_VEL
LIN {X 0,Y 452.861,Z 388.292,A -85,B 0,C 180,E1 -8385.806,E2 -8385.806} C_VEL
LIN {X 0,Y 453.074,Z 379.663,A -85,B 0,C 180,E1 -8389.012,E2 -8389.012} C_VEL
LIN {X 0,Y 453.307,Z 372.209,A -85,B 0,C 180,E1 -8391.846,E2 -8391.846} C_VEL
LIN {X 0,Y 453.672,Z 363.564,A -85,B 0,C 180,E1 -8395.216,E2 -8395.216} C_VEL
LIN {X 0,Y 454.121,Z 355.112,A -85,B 0,C 180,E1 -8398.671,E2 -8398.671} C_VEL
LIN {X 0,Y 454.528,Z 349.149,A -85,B 0,C 180,E1 -8401.198,E2 -8401.198} C_VEL
LIN {X 0,Y 454.775,Z 345.621,A -85,B 0,C 180,E1 -8402.745,E2 -8402.745} C_VEL
LIN {X 0,Y 454.415,Z 342.145,A -85,B 0,C 180,E1 -8404.362,E2 -8404.362} C_VEL
LIN {X 0,Y 453.479,Z 336.813,A -85,B 0,C 180,E1 -8407.073,E2 -8407.073} C_VEL
LIN {X 0,Y 453.511,Z 336.813,A -85,B 0,C 180,E1 -8409.449,E2 -8409.449} C_VEL
LIN {X 0,Y 453.469,Z 336.819,A -85,B 0,C 180,E1 -8412.995,E2 -8412.995} C_VEL
LIN {X 0,Y 453.468,Z 336.815,A -85,B 0,C 180,E1 -8415.779,E2 -8415.779} C_VEL
LIN {X 0,Y 453.486,Z 336.811,A -85,B 0,C 180,E1 -8418.209,E2 -8418.209} C_VEL
LIN {X 0,Y 453.477,Z 336.812,A -85,B 0,C 180,E1 -8420.797,E2 -8420.797} C_VEL
LIN {X 0,Y 453.46,Z 336.814,A -85,B 0,C 180,E1 -8423.917,E2 -8423.917} C_VEL
LIN {X 0,Y 453.485,Z 336.812,A -85,B 0,C 180,E1 -8427.151,E2 -8427.151} C_VEL
LIN {X 0,Y 453.48,Z 336.812,A -85,B 0,C 180,E1 -8430.268,E2 -8430.268} C_VEL
LIN {X 0,Y 453.511,Z 336.808,A -85,B 0,C 180,E1 -8433.294,E2 -8433.294} C_VEL
LIN {X 0,Y 453.509,Z 336.809,A -85,B 0,C 180,E1 -8436.238,E2 -8436.238} C_VEL
LIN {X 0,Y 453.489,Z 336.811,A -85,B 0,C 180,E1 -8439.117,E2 -8439.117} C_VEL
LIN {X 0,Y 453.51,Z 336.807,A -85,B 0,C 180,E1 -8441.944,E2 -8441.944} C_VEL
LIN {X 0,Y 453.546,Z 336.805,A -85,B 0,C 180,E1 -8444.726,E2 -8444.726} C_VEL
LIN {X 0,Y 453.565,Z 336.802,A -85,B 0,C 180,E1 -8448.378,E2 -8448.378} C_VEL
LIN {X 0,Y 453.591,Z 336.798,A -85,B 0,C 180,E1 -8451.086,E2 -8451.086} C_VEL
LIN {X 0,Y 453.657,Z 336.789,A -85,B 0,C 180,E1 -8453.774,E2 -8453.774} C_VEL
LIN {X 0,Y 453.74,Z 336.779,A -85,B 0,C 180,E1 -8457.336,E2 -8457.336} C_VEL
LIN {X 0,Y 453.828,Z 336.77,A -85,B 0,C 180,E1 -8459.999,E2 -8459.999} C_VEL
LIN {X 0,Y 453.747,Z 336.778,A -85,B 0,C 180,E1 -8462.662,E2 -8462.662} C_VEL
LIN {X 0,Y 453.673,Z 336.789,A -85,B 0,C 180,E1 -8466.224,E2 -8466.224} C_VEL
LIN {X 0,Y 453.589,Z 336.798,A -85,B 0,C 180,E1 -8468.912,E2 -8468.912} C_VEL
LIN {X 0,Y 453.568,Z 336.801,A -85,B 0,C 180,E1 -8472.528,E2 -8472.528} C_VEL
LIN {X 0,Y 453.538,Z 336.808,A -85,B 0,C 180,E1 -8476.195,E2 -8476.195} C_VEL
LIN {X 0,Y 453.27,Z 336.84,A -85,B 0,C 180,E1 -8479.001,E2 -8479.001} C_VEL
LIN {X 0,Y 453.119,Z 337.302,A -85,B 0,C 180,E1 -8479.95,E2 -8479.95} C_VEL
LIN {X 0,Y 453.014,Z 340.712,A -85,B 0,C 180,E1 -8482.819,E2 -8482.819} C_VEL
LIN {X 0,Y 452.901,Z 344.352,A -85,B 0,C 180,E1 -8485.837,E2 -8485.837} C_VEL
LIN {X 0,Y 452.83,Z 347.936,A -85,B 0,C 180,E1 -8488.758,E2 -8488.758} C_VEL
LIN {X 0,Y 452.72,Z 351.815,A -85,B 0,C 180,E1 -8491.856,E2 -8491.856} C_VEL
LIN {X 0,Y 452.619,Z 355.896,A -85,B 0,C 180,E1 -8495.064,E2 -8495.064} C_VEL
LIN {X 0,Y 452.603,Z 359.099,A -85,B 0,C 180,E1 -8497.563,E2 -8497.563} C_VEL
LIN {X 0,Y 454.773,Z 370.57,A -85,B 0,C 180,E1 -8498.076,E2 -8498.076} C_VEL
LIN {X 0,Y 454.962,Z 376.488,A -85,B 0,C 180,E1 -8498.373,E2 -8498.373} C_VEL
LIN {X 0,Y 454.629,Z 386.918,A -85,B 0,C 180,E1 -8499.044,E2 -8499.044} C_VEL
LIN {X 0,Y 454.291,Z 394.442,A -85,B 0,C 180,E1 -8499.652,E2 -8499.652} C_VEL
LIN {X 0,Y 454.004,Z 402.068,A -85,B 0,C 180,E1 -8500.406,E2 -8500.406} C_VEL
LIN {X 0,Y 453.687,Z 408.571,A -85,B 0,C 180,E1 -8501.181,E2 -8501.181} C_VEL
LIN {X 0,Y 453.472,Z 413.897,A -85,B 0,C 180,E1 -8501.933,E2 -8501.933} C_VEL
LIN {X 0,Y 453.153,Z 420.282,A -85,B 0,C 180,E1 -8503.03,E2 -8503.03} C_VEL
LIN {X 0,Y 452.958,Z 424.832,A -85,B 0,C 180,E1 -8503.995,E2 -8503.995} C_VEL
LIN {X 0,Y 452.778,Z 428.809,A -85,B 0,C 180,E1 -8505.042,E2 -8505.042} C_VEL
LIN {X 0,Y 452.732,Z 430.876,A -85,B 0,C 180,E1 -8505.687,E2 -8505.687} C_VEL
LIN {X 0,Y 452.564,Z 433.777,A -85,B 0,C 180,E1 -8506.898,E2 -8506.898} C_VEL
LIN {X 0,Y 452.467,Z 435.792,A -85,B 0,C 180,E1 -8508.206,E2 -8508.206} C_VEL
LIN {X 0,Y 452.393,Z 436.752,A -85,B 0,C 180,E1 -8509.57,E2 -8509.57} C_VEL
LIN {X 0,Y 452.4,Z 436.561,A -85,B 0,C 180,E1 -8510.961,E2 -8510.961} C_VEL
LIN {X 0,Y 452.471,Z 435.096,A -85,B 0,C 180,E1 -8512.385,E2 -8512.385} C_VEL
LIN {X 0,Y 452.595,Z 432.105,A -85,B 0,C 180,E1 -8513.847,E2 -8513.847} C_VEL
LIN {X 0,Y 452.719,Z 428.912,A -85,B 0,C 180,E1 -8514.942,E2 -8514.942} C_VEL
LIN {X 0,Y 452.919,Z 424.75,A -85,B 0,C 180,E1 -8516.039,E2 -8516.039} C_VEL
LIN {X 0,Y 453.12,Z 419.576,A -85,B 0,C 180,E1 -8517.121,E2 -8517.121} C_VEL
LIN {X 0,Y 453.439,Z 413.16,A -85,B 0,C 180,E1 -8518.198,E2 -8518.198} C_VEL
LIN {X 0,Y 453.836,Z 404.213,A -85,B 0,C 180,E1 -8519.377,E2 -8519.377} C_VEL
LIN {X 0,Y 454.096,Z 396.721,A -85,B 0,C 180,E1 -8520.161,E2 -8520.161} C_VEL
LIN {X 0,Y 454.409,Z 388.748,A -85,B 0,C 180,E1 -8520.843,E2 -8520.843} C_VEL
LIN {X 0,Y 454.659,Z 381.282,A -85,B 0,C 180,E1 -8521.366,E2 -8521.366} C_VEL
LIN {X 0,Y 454.933,Z 371.763,A -85,B 0,C 180,E1 -8521.888,E2 -8521.888} C_VEL
LIN {X 0,Y 453.325,Z 362.669,A -85,B 0,C 180,E1 -8522.308,E2 -8522.308} C_VEL
LIN {X 0,Y 452.616,Z 358.553,A -85,B 0,C 180,E1 -8522.486,E2 -8522.486} C_VEL
LIN {X 0,Y 452.61,Z 354.956,A -85,B 0,C 180,E1 -8525.212,E2 -8525.212} C_VEL
LIN {X 0,Y 452.656,Z 350.44,A -85,B 0,C 180,E1 -8528.676,E2 -8528.676} C_VEL
LIN {X 0,Y 452.77,Z 346.297,A -85,B 0,C 180,E1 -8531.913,E2 -8531.913} C_VEL
LIN {X 0,Y 452.774,Z 345.363,A -85,B 0,C 180,E1 -8532.642,E2 -8532.642} C_VEL
LIN {X 0,Y 452.145,Z 344.49,A -85,B 0,C 180,E1 -8533.376,E2 -8533.376} C_VEL
LIN {X 0,Y 449.317,Z 343.26,A -85,B 0,C 180,E1 -8534.573,E2 -8534.573} C_VEL
LIN {X 0,Y 446.916,Z 342.296,A -85,B 0,C 180,E1 -8535.539,E2 -8535.539} C_VEL
LIN {X 0,Y 445.899,Z 341.477,A -85,B 0,C 180,E1 -8536.284,E2 -8536.284} C_VEL
LIN {X 0,Y 445.825,Z 341.169,A -85,B 0,C 180,E1 -8536.535,E2 -8536.535} C_VEL
LIN {X 0,Y 445.973,Z 338.01,A -85,B 0,C 180,E1 -8539.098,E2 -8539.098} C_VEL
LIN {X 0,Y 446.382,Z 337.697,A -85,B 0,C 180,E1 -8541.853,E2 -8541.853} C_VEL
LIN {X 0,Y 446.63,Z 337.666,A -85,B 0,C 180,E1 -8544.581,E2 -8544.581} C_VEL
LIN {X 0,Y 446.699,Z 337.655,A -85,B 0,C 180,E1 -8547.294,E2 -8547.294} C_VEL
LIN {X 0,Y 446.783,Z 337.647,A -85,B 0,C 180,E1 -8549.999,E2 -8549.999} C_VEL
LIN {X 0,Y 446.7,Z 337.655,A -85,B 0,C 180,E1 -8552.704,E2 -8552.704} C_VEL
LIN {X 0,Y 446.641,Z 337.664,A -85,B 0,C 180,E1 -8556.323,E2 -8556.323} C_VEL
LIN {X 0,Y 446.528,Z 337.676,A -85,B 0,C 180,E1 -8559.054,E2 -8559.054} C_VEL
LIN {X 0,Y 446.521,Z 337.677,A -85,B 0,C 180,E1 -8562.728,E2 -8562.728} C_VEL
LIN {X 0,Y 446.477,Z 337.683,A -85,B 0,C 180,E1 -8566.458,E2 -8566.458} C_VEL
LIN {X 0,Y 446.456,Z 337.688,A -85,B 0,C 180,E1 -8569.302,E2 -8569.302} C_VEL
LIN {X 0,Y 446.404,Z 337.693,A -85,B 0,C 180,E1 -8572.199,E2 -8572.199} C_VEL
LIN {X 0,Y 446.444,Z 337.688,A -85,B 0,C 180,E1 -8575.152,E2 -8575.152} C_VEL
LIN {X 0,Y 446.47,Z 337.684,A -85,B 0,C 180,E1 -8578.178,E2 -8578.178} C_VEL
LIN {X 0,Y 446.406,Z 337.695,A -85,B 0,C 180,E1 -8581.299,E2 -8581.299} C_VEL
LIN {X 0,Y 446.416,Z 337.689,A -85,B 0,C 180,E1 -8584.522,E2 -8584.522} C_VEL
LIN {X 0,Y 446.424,Z 337.689,A -85,B 0,C 180,E1 -8588.083,E2 -8588.083} C_VEL
LIN {X 0,Y 446.433,Z 337.691,A -85,B 0,C 180,E1 -8590.921,E2 -8590.921} C_VEL
LIN {X 0,Y 446.43,Z 337.688,A -85,B 0,C 180,E1 -8593.84,E2 -8593.84} C_VEL
LIN {X 0,Y 446.432,Z 337.689,A -85,B 0,C 180,E1 -8596.397,E2 -8596.397} C_VEL
LIN {X 0,Y 446.454,Z 337.684,A -85,B 0,C 180,E1 -8599.805,E2 -8599.805} C_VEL
LIN {X 0,Y 446.42,Z 337.69,A -85,B 0,C 180,E1 -8602.124,E2 -8602.124} C_VEL
LIN {X 0,Y 446.416,Z 337.691,A -85,B 0,C 180,E1 -8605.477,E2 -8605.477} C_VEL
LIN {X 0,Y 446.405,Z 337.693,A -85,B 0,C 180,E1 -8608.7,E2 -8608.7} C_VEL
LIN {X 0,Y 446.47,Z 337.684,A -85,B 0,C 180,E1 -8611.822,E2 -8611.822} C_VEL
LIN {X 0,Y 446.445,Z 337.689,A -85,B 0,C 180,E1 -8614.848,E2 -8614.848} C_VEL
LIN {X 0,Y 446.458,Z 337.686,A -85,B 0,C 180,E1 -8618.238,E2 -8618.238} C_VEL
LIN {X 0,Y 446.444,Z 337.687,A -85,B 0,C 180,E1 -8621.65,E2 -8621.65} C_VEL
LIN {X 0,Y 446.503,Z 337.681,A -85,B 0,C 180,E1 -8624.481,E2 -8624.481} C_VEL
LIN {X 0,Y 446.526,Z 337.678,A -85,B 0,C 180,E1 -8628.194,E2 -8628.194} C_VEL
LIN {X 0,Y 446.588,Z 337.67,A -85,B 0,C 180,E1 -8631.859,E2 -8631.859} C_VEL
LIN {X 0,Y 446.635,Z 337.664,A -85,B 0,C 180,E1 -8634.583,E2 -8634.583} C_VEL
LIN {X 0,Y 446.699,Z 337.656,A -85,B 0,C 180,E1 -8637.296,E2 -8637.296} C_VEL
LIN {X 0,Y 446.782,Z 337.646,A -85,B 0,C 180,E1 -8640.001,E2 -8640.001} C_VEL
LIN {X 0,Y 446.701,Z 337.655,A -85,B 0,C 180,E1 -8642.706,E2 -8642.706} C_VEL
LIN {X 0,Y 446.636,Z 337.664,A -85,B 0,C 180,E1 -8646.325,E2 -8646.325} C_VEL
LIN {X 0,Y 446.529,Z 337.676,A -85,B 0,C 180,E1 -8649.056,E2 -8649.056} C_VEL
LIN {X 0,Y 446.524,Z 337.677,A -85,B 0,C 180,E1 -8652.73,E2 -8652.73} C_VEL
LIN {X 0,Y 446.48,Z 337.682,A -85,B 0,C 180,E1 -8656.46,E2 -8656.46} C_VEL
LIN {X 0,Y 446.46,Z 337.687,A -85,B 0,C 180,E1 -8659.304,E2 -8659.304} C_VEL
LIN {X 0,Y 446.409,Z 337.691,A -85,B 0,C 180,E1 -8662.201,E2 -8662.201} C_VEL
LIN {X 0,Y 446.45,Z 337.689,A -85,B 0,C 180,E1 -8665.153,E2 -8665.153} C_VEL
LIN {X 0,Y 446.476,Z 337.682,A -85,B 0,C 180,E1 -8668.18,E2 -8668.18} C_VEL
LIN {X 0,Y 446.412,Z 337.693,A -85,B 0,C 180,E1 -8671.301,E2 -8671.301} C_VEL
LIN {X 0,Y 446.423,Z 337.689,A -85,B 0,C 180,E1 -8674.524,E2 -8674.524} C_VEL
LIN {X 0,Y 446.424,Z 337.689,A -85,B 0,C 180,E1 -8678.083,E2 -8678.083} C_VEL
LIN {X 0,Y 446.421,Z 337.692,A -85,B 0,C 180,E1 -8680.919,E2 -8680.919} C_VEL
LIN {X 0,Y 446.417,Z 337.689,A -85,B 0,C 180,E1 -8683.845,E2 -8683.845} C_VEL
LIN {X 0,Y 446.415,Z 337.691,A -85,B 0,C 180,E1 -8686.402,E2 -8686.402} C_VEL
LIN {X 0,Y 446.446,Z 337.687,A -85,B 0,C 180,E1 -8689.804,E2 -8689.804} C_VEL
LIN {X 0,Y 446.445,Z 337.69,A -85,B 0,C 180,E1 -8693.12,E2 -8693.12} C_VEL
LIN {X 0,Y 447.399,Z 342.891,A -85,B 0,C 180,E1 -8695.564,E2 -8695.564} C_VEL
LIN {X 0,Y 447.728,Z 346.566,A -85,B 0,C 180,E1 -8697.213,E2 -8697.213} C_VEL
LIN {X 0,Y 447.274,Z 353.922,A -85,B 0,C 180,E1 -8700.335,E2 -8700.335} C_VEL
LIN {X 0,Y 446.784,Z 362.167,A -85,B 0,C 180,E1 -8703.718,E2 -8703.718} C_VEL
LIN {X 0,Y 446.403,Z 369.959,A -85,B 0,C 180,E1 -8706.823,E2 -8706.823} C_VEL
LIN {X 0,Y 446.099,Z 378.632,A -85,B 0,C 180,E1 -8710.203,E2 -8710.203} C_VEL
LIN {X 0,Y 445.844,Z 387.326,A -85,B 0,C 180,E1 -8713.518,E2 -8713.518} C_VEL
LIN {X 0,Y 445.606,Z 396.038,A -85,B 0,C 180,E1 -8716.781,E2 -8716.781} C_VEL
LIN {X 0,Y 445.6,Z 397.451,A -85,B 0,C 180,E1 -8717.308,E2 -8717.308} C_VEL
LIN {X 0,Y 446.942,Z 410.26,A -85,B 0,C 180,E1 -8717.79,E2 -8717.79} C_VEL
LIN {X 0,Y 447.546,Z 418.605,A -85,B 0,C 180,E1 -8718.222,E2 -8718.222} C_VEL
LIN {X 0,Y 447.224,Z 427.449,A -85,B 0,C 180,E1 -8718.788,E2 -8718.788} C_VEL
LIN {X 0,Y 446.832,Z 435.878,A -85,B 0,C 180,E1 -8719.466,E2 -8719.466} C_VEL
LIN {X 0,Y 446.475,Z 443.85,A -85,B 0,C 180,E1 -8720.259,E2 -8720.259} C_VEL
LIN {X 0,Y 446.243,Z 449.592,A -85,B 0,C 180,E1 -8720.94,E2 -8720.94} C_VEL
LIN {X 0,Y 445.955,Z 456.008,A -85,B 0,C 180,E1 -8721.847,E2 -8721.847} C_VEL
LIN {X 0,Y 445.755,Z 461.345,A -85,B 0,C 180,E1 -8722.755,E2 -8722.755} C_VEL
LIN {X 0,Y 445.577,Z 465.796,A -85,B 0,C 180,E1 -8723.662,E2 -8723.662} C_VEL
LIN {X 0,Y 445.513,Z 471.034,A -85,B 0,C 180,E1 -8725.024,E2 -8725.024} C_VEL
LIN {X 0,Y 445.414,Z 473.719,A -85,B 0,C 180,E1 -8725.93,E2 -8725.93} C_VEL
LIN {X 0,Y 445.459,Z 476.659,A -85,B 0,C 180,E1 -8727.288,E2 -8727.288} C_VEL
LIN {X 0,Y 445.399,Z 477.93,A -85,B 0,C 180,E1 -8728.193,E2 -8728.193} C_VEL
LIN {X 0,Y 445.393,Z 478.723,A -85,B 0,C 180,E1 -8729.097,E2 -8729.097} C_VEL
LIN {X 0,Y 445.4,Z 479.013,A -85,B 0,C 180,E1 -8730.001,E2 -8730.001} C_VEL
LIN {X 0,Y 445.393,Z 478.708,A -85,B 0,C 180,E1 -8730.905,E2 -8730.905} C_VEL
LIN {X 0,Y 445.4,Z 477.919,A -85,B 0,C 180,E1 -8731.81,E2 -8731.81} C_VEL
LIN {X 0,Y 445.459,Z 476.65,A -85,B 0,C 180,E1 -8732.714,E2 -8732.714} C_VEL
LIN {X 0,Y 445.413,Z 473.702,A -85,B 0,C 180,E1 -8734.073,E2 -8734.073} C_VEL
LIN {X 0,Y 445.514,Z 471.026,A -85,B 0,C 180,E1 -8734.979,E2 -8734.979} C_VEL
LIN {X 0,Y 445.579,Z 465.783,A -85,B 0,C 180,E1 -8736.34,E2 -8736.34} C_VEL
LIN {X 0,Y 445.855,Z 458.898,A -85,B 0,C 180,E1 -8737.701,E2 -8737.701} C_VEL
LIN {X 0,Y 446.141,Z 451.381,A -85,B 0,C 180,E1 -8738.836,E2 -8738.836} C_VEL
LIN {X 0,Y 446.487,Z 443.982,A -85,B 0,C 180,E1 -8739.743,E2 -8739.743} C_VEL
LIN {X 0,Y 446.84,Z 436.077,A -85,B 0,C 180,E1 -8740.536,E2 -8740.536} C_VEL
LIN {X 0,Y 447.235,Z 427.752,A -85,B 0,C 180,E1 -8741.215,E2 -8741.215} C_VEL
LIN {X 0,Y 447.63,Z 417.348,A -85,B 0,C 180,E1 -8741.883,E2 -8741.883} C_VEL
LIN {X 0,Y 446.609,Z 405.658,A -85,B 0,C 180,E1 -8742.445,E2 -8742.445} C_VEL
LIN {X 0,Y 445.586,Z 396.889,A -85,B 0,C 180,E1 -8742.758,E2 -8742.758} C_VEL
LIN {X 0,Y 445.774,Z 388.433,A -85,B 0,C 180,E1 -8745.905,E2 -8745.905} C_VEL
LIN {X 0,Y 446.02,Z 379.419,A -85,B 0,C 180,E1 -8749.324,E2 -8749.324} C_VEL
LIN {X 0,Y 446.27,Z 371.98,A -85,B 0,C 180,E1 -8752.208,E2 -8752.208} C_VEL
LIN {X 0,Y 446.697,Z 363.432,A -85,B 0,C 180,E1 -8755.638,E2 -8755.638} C_VEL
LIN {X 0,Y 447.095,Z 356.11,A -85,B 0,C 180,E1 -8758.684,E2 -8758.684} C_VEL
LIN {X 0,Y 447.53,Z 350.245,A -85,B 0,C 180,E1 -8761.215,E2 -8761.215} C_VEL
LIN {X 0,Y 447.71,Z 345.578,A -85,B 0,C 180,E1 -8763.328,E2 -8763.328} C_VEL
LIN {X 0,Y 446.83,Z 339.944,A -85,B 0,C 180,E1 -8766.099,E2 -8766.099} C_VEL
LIN {X 0,Y 446.426,Z 337.692,A -85,B 0,C 180,E1 -8767.309,E2 -8767.309} C_VEL
LIN {X 0,Y 446.454,Z 337.692,A -85,B 0,C 180,E1 -8770.198,E2 -8770.198} C_VEL
LIN {X 0,Y 446.436,Z 337.695,A -85,B 0,C 180,E1 -8772.605,E2 -8772.605} C_VEL
LIN {X 0,Y 446.458,Z 337.691,A -85,B 0,C 180,E1 -8775.104,E2 -8775.104} C_VEL
LIN {X 0,Y 446.435,Z 337.691,A -85,B 0,C 180,E1 -8778.609,E2 -8778.609} C_VEL
LIN {X 0,Y 446.419,Z 337.691,A -85,B 0,C 180,E1 -8781.921,E2 -8781.921} C_VEL
LIN {X 0,Y 446.43,Z 337.69,A -85,B 0,C 180,E1 -8785.476,E2 -8785.476} C_VEL
LIN {X 0,Y 446.422,Z 337.69,A -85,B 0,C 180,E1 -8788.699,E2 -8788.699} C_VEL
LIN {X 0,Y 446.492,Z 337.684,A -85,B 0,C 180,E1 -8791.821,E2 -8791.821} C_VEL
LIN {X 0,Y 446.457,Z 337.686,A -85,B 0,C 180,E1 -8794.847,E2 -8794.847} C_VEL
LIN {X 0,Y 446.455,Z 337.686,A -85,B 0,C 180,E1 -8798.245,E2 -8798.245} C_VEL
LIN {X 0,Y 446.458,Z 337.686,A -85,B 0,C 180,E1 -8801.649,E2 -8801.649} C_VEL
LIN {X 0,Y 446.514,Z 337.68,A -85,B 0,C 180,E1 -8804.479,E2 -8804.479} C_VEL
LIN {X 0,Y 446.523,Z 337.679,A -85,B 0,C 180,E1 -8808.192,E2 -8808.192} C_VEL
LIN {X 0,Y 446.538,Z 337.677,A -85,B 0,C 180,E1 -8810.944,E2 -8810.944} C_VEL
LIN {X 0,Y 446.625,Z 337.665,A -85,B 0,C 180,E1 -8813.675,E2 -8813.675} C_VEL
LIN {X 0,Y 446.687,Z 337.658,A -85,B 0,C 180,E1 -8817.294,E2 -8817.294} C_VEL
LIN {X 0,Y 446.798,Z 337.646,A -85,B 0,C 180,E1 -8819.999,E2 -8819.999} C_VEL
LIN {X 0,Y 446.694,Z 337.657,A -85,B 0,C 180,E1 -8822.704,E2 -8822.704} C_VEL
LIN {X 0,Y 446.642,Z 337.664,A -85,B 0,C 180,E1 -8826.323,E2 -8826.323} C_VEL
LIN {X 0,Y 446.536,Z 337.676,A -85,B 0,C 180,E1 -8829.054,E2 -8829.054} C_VEL
LIN {X 0,Y 446.525,Z 337.679,A -85,B 0,C 180,E1 -8832.729,E2 -8832.729} C_VEL
LIN {X 0,Y 446.511,Z 337.684,A -85,B 0,C 180,E1 -8836.232,E2 -8836.232} C_VEL
LIN {X 0,Y 446.148,Z 337.727,A -85,B 0,C 180,E1 -8839.316,E2 -8839.316} C_VEL
LIN {X 0,Y 446.023,Z 340.105,A -85,B 0,C 180,E1 -8841.616,E2 -8841.616} C_VEL
LIN {X 0,Y 445.951,Z 343.144,A -85,B 0,C 180,E1 -8844.188,E2 -8844.188} C_VEL
LIN {X 0,Y 445.782,Z 346.803,A -85,B 0,C 180,E1 -8847.205,E2 -8847.205} C_VEL
LIN {X 0,Y 445.701,Z 350.609,A -85,B 0,C 180,E1 -8850.303,E2 -8850.303} C_VEL
LIN {X 0,Y 445.598,Z 354.577,A -85,B 0,C 180,E1 -8853.504,E2 -8853.504} C_VEL
LIN {X 0,Y 445.498,Z 358.775,A -85,B 0,C 180,E1 -8856.831,E2 -8856.831} C_VEL
LIN {X 0,Y 445.521,Z 359.515,A -85,B 0,C 180,E1 -8857.359,E2 -8857.359} C_VEL
LIN {X 0,Y 447.644,Z 370.595,A -85,B 0,C 180,E1 -8857.858,E2 -8857.858} C_VEL
LIN {X 0,Y 448.108,Z 374.507,A -85,B 0,C 180,E1 -8858.062,E2 -8858.062} C_VEL
LIN {X 0,Y 447.717,Z 385.861,A -85,B 0,C 180,E1 -8858.757,E2 -8858.757} C_VEL
LIN {X 0,Y 447.345,Z 394.758,A -85,B 0,C 180,E1 -8859.48,E2 -8859.48} C_VEL
LIN {X 0,Y 447.037,Z 401.375,A -85,B 0,C 180,E1 -8860.132,E2 -8860.132} C_VEL
LIN {X 0,Y 446.697,Z 408.327,A -85,B 0,C 180,E1 -8860.956,E2 -8860.956} C_VEL
LIN {X 0,Y 446.442,Z 414.346,A -85,B 0,C 180,E1 -8861.816,E2 -8861.816} C_VEL
LIN {X 0,Y 446.159,Z 420.316,A -85,B 0,C 180,E1 -8862.854,E2 -8862.854} C_VEL
LIN {X 0,Y 445.917,Z 425.218,A -85,B 0,C 180,E1 -8863.904,E2 -8863.904} C_VEL
LIN {X 0,Y 445.748,Z 428.644,A -85,B 0,C 180,E1 -8864.804,E2 -8864.804} C_VEL
LIN {X 0,Y 445.572,Z 432.319,A -85,B 0,C 180,E1 -8866.05,E2 -8866.05} C_VEL
LIN {X 0,Y 445.432,Z 434.881,A -85,B 0,C 180,E1 -8867.276,E2 -8867.276} C_VEL
LIN {X 0,Y 445.366,Z 436.459,A -85,B 0,C 180,E1 -8868.487,E2 -8868.487} C_VEL
LIN {X 0,Y 445.298,Z 437.127,A -85,B 0,C 180,E1 -8869.676,E2 -8869.676} C_VEL
LIN {X 0,Y 445.315,Z 436.936,A -85,B 0,C 180,E1 -8870.854,E2 -8870.854} C_VEL
LIN {X 0,Y 445.354,Z 435.834,A -85,B 0,C 180,E1 -8872.093,E2 -8872.093} C_VEL
LIN {X 0,Y 445.509,Z 433.287,A -85,B 0,C 180,E1 -8873.563,E2 -8873.563} C_VEL
LIN {X 0,Y 445.672,Z 428.996,A -85,B 0,C 180,E1 -8875.083,E2 -8875.083} C_VEL
LIN {X 0,Y 445.887,Z 424.561,A -85,B 0,C 180,E1 -8876.247,E2 -8876.247} C_VEL
LIN {X 0,Y 446.124,Z 419.119,A -85,B 0,C 180,E1 -8877.374,E2 -8877.374} C_VEL
LIN {X 0,Y 446.473,Z 412.523,A -85,B 0,C 180,E1 -8878.469,E2 -8878.469} C_VEL
LIN {X 0,Y 446.827,Z 404.502,A -85,B 0,C 180,E1 -8879.518,E2 -8879.518} C_VEL
LIN {X 0,Y 447.118,Z 396.938,A -85,B 0,C 180,E1 -8880.321,E2 -8880.321} C_VEL
LIN {X 0,Y 447.456,Z 388.548,A -85,B 0,C 180,E1 -8881.043,E2 -8881.043} C_VEL
LIN {X 0,Y 447.789,Z 380.385,A -85,B 0,C 180,E1 -8881.608,E2 -8881.608} C_VEL
LIN {X 0,Y 447.974,Z 372.918,A -85,B 0,C 180,E1 -8882.025,E2 -8882.025} C_VEL
LIN {X 0,Y 446.307,Z 363.28,A -85,B 0,C 180,E1 -8882.484,E2 -8882.484} C_VEL
LIN {X 0,Y 445.544,Z 358.873,A -85,B 0,C 180,E1 -8882.662,E2 -8882.662} C_VEL
LIN {X 0,Y 445.568,Z 354.276,A -85,B 0,C 180,E1 -8886.179,E2 -8886.179} C_VEL
LIN {X 0,Y 445.608,Z 349.755,A -85,B 0,C 180,E1 -8889.696,E2 -8889.696} C_VEL
LIN {X 0,Y 445.71,Z 346.004,A -85,B 0,C 180,E1 -8892.654,E2 -8892.654} C_VEL
LIN {X 0,Y 445.779,Z 342.593,A -85,B 0,C 180,E1 -8895.388,E2 -8895.388} C_VEL
LIN {X 0,Y 445.825,Z 341.169,A -85,B 0,C 180,E1 -8896.535,E2 -8896.535} C_VEL
LIN {X 0,Y 445.185,Z 340.313,A -85,B 0,C 180,E1 -8897.282,E2 -8897.282} C_VEL
LIN {X 0,Y 442.385,Z 339.272,A -85,B 0,C 180,E1 -8898.504,E2 -8898.504} C_VEL
LIN {X 0,Y 440.067,Z 338.783,A -85,B 0,C 180,E1 -8899.493,E2 -8899.493} C_VEL
LIN {X 0,Y 439.156,Z 338.616,A -85,B 0,C 180,E1 -8900.257,E2 -8900.257} C_VEL
LIN {X 0,Y 439.127,Z 338.599,A -85,B 0,C 180,E1 -8900.516,E2 -8900.516} C_VEL
LIN {X 0,Y 439.513,Z 338.551,A -85,B 0,C 180,E1 -8902.649,E2 -8902.649} C_VEL
LIN {X 0,Y 439.604,Z 338.541,A -85,B 0,C 180,E1 -8904.494,E2 -8904.494} C_VEL
LIN {X 0,Y 439.626,Z 338.538,A -85,B 0,C 180,E1 -8908.167,E2 -8908.167} C_VEL
LIN {X 0,Y 439.753,Z 338.522,A -85,B 0,C 180,E1 -8909.999,E2 -8909.999} C_VEL
LIN {X 0,Y 439.647,Z 338.534,A -85,B 0,C 180,E1 -8912.748,E2 -8912.748} C_VEL
LIN {X 0,Y 439.611,Z 338.539,A -85,B 0,C 180,E1 -8916.424,E2 -8916.424} C_VEL
LIN {X 0,Y 439.49,Z 338.553,A -85,B 0,C 180,E1 -8919.201,E2 -8919.201} C_VEL
LIN {X 0,Y 439.491,Z 338.553,A -85,B 0,C 180,E1 -8922.726,E2 -8922.726} C_VEL
LIN {X 0,Y 439.434,Z 338.561,A -85,B 0,C 180,E1 -8926.348,E2 -8926.348} C_VEL
LIN {X 0,Y 439.389,Z 338.567,A -85,B 0,C 180,E1 -8929.625,E2 -8929.625} C_VEL
LIN {X 0,Y 439.351,Z 338.57,A -85,B 0,C 180,E1 -8932.575,E2 -8932.575} C_VEL
LIN {X 0,Y 439.392,Z 338.567,A -85,B 0,C 180,E1 -8935.584,E2 -8935.584} C_VEL
LIN {X 0,Y 439.411,Z 338.563,A -85,B 0,C 180,E1 -8938.672,E2 -8938.672} C_VEL
LIN {X 0,Y 439.36,Z 338.57,A -85,B 0,C 180,E1 -8941.86,E2 -8941.86} C_VEL
LIN {X 0,Y 439.386,Z 338.568,A -85,B 0,C 180,E1 -8945.155,E2 -8945.155} C_VEL
LIN {X 0,Y 439.385,Z 338.567,A -85,B 0,C 180,E1 -8948.593,E2 -8948.593} C_VEL
LIN {X 0,Y 439.39,Z 338.567,A -85,B 0,C 180,E1 -8951.259,E2 -8951.259} C_VEL
LIN {X 0,Y 439.395,Z 338.567,A -85,B 0,C 180,E1 -8954.728,E2 -8954.728} C_VEL
LIN {X 0,Y 439.397,Z 338.564,A -85,B 0,C 180,E1 -8957.798,E2 -8957.798} C_VEL
LIN {X 0,Y 439.437,Z 338.559,A -85,B 0,C 180,E1 -8960.23,E2 -8960.23} C_VEL
LIN {X 0,Y 439.363,Z 338.568,A -85,B 0,C 180,E1 -8963.713,E2 -8963.713} C_VEL
LIN {X 0,Y 439.36,Z 338.57,A -85,B 0,C 180,E1 -8967.055,E2 -8967.055} C_VEL
LIN {X 0,Y 439.382,Z 338.567,A -85,B 0,C 180,E1 -8970.276,E2 -8970.276} C_VEL
LIN {X 0,Y 439.419,Z 338.561,A -85,B 0,C 180,E1 -8973.589,E2 -8973.589} C_VEL
LIN {X 0,Y 439.378,Z 338.57,A -85,B 0,C 180,E1 -8976.43,E2 -8976.43} C_VEL
LIN {X 0,Y 439.392,Z 338.564,A -85,B 0,C 180,E1 -8979.399,E2 -8979.399} C_VEL
LIN {X 0,Y 439.419,Z 338.564,A -85,B 0,C 180,E1 -8982.31,E2 -8982.31} C_VEL
LIN {X 0,Y 439.438,Z 338.559,A -85,B 0,C 180,E1 -8985.175,E2 -8985.175} C_VEL
LIN {X 0,Y 439.495,Z 338.554,A -85,B 0,C 180,E1 -8988.003,E2 -8988.003} C_VEL
LIN {X 0,Y 439.536,Z 338.548,A -85,B 0,C 180,E1 -8991.727,E2 -8991.727} C_VEL
LIN {X 0,Y 439.61,Z 338.54,A -85,B 0,C 180,E1 -8994.497,E2 -8994.497} C_VEL
LIN {X 0,Y 439.624,Z 338.539,A -85,B 0,C 180,E1 -8998.169,E2 -8998.169} C_VEL
LIN {X 0,Y 439.752,Z 338.522,A -85,B 0,C 180,E1 -9000.001,E2 -9000.001} C_VEL
LIN {X 0,Y 439.647,Z 338.533,A -85,B 0,C 180,E1 -9002.75,E2 -9002.75} C_VEL
LIN {X 0,Y 439.607,Z 338.539,A -85,B 0,C 180,E1 -9006.426,E2 -9006.426} C_VEL
LIN {X 0,Y 439.491,Z 338.554,A -85,B 0,C 180,E1 -9009.203,E2 -9009.203} C_VEL
LIN {X 0,Y 439.494,Z 338.552,A -85,B 0,C 180,E1 -9012.728,E2 -9012.728} C_VEL
LIN {X 0,Y 439.438,Z 338.56,A -85,B 0,C 180,E1 -9016.35,E2 -9016.35} C_VEL
LIN {X 0,Y 439.393,Z 338.567,A -85,B 0,C 180,E1 -9019.627,E2 -9019.627} C_VEL
LIN {X 0,Y 439.356,Z 338.57,A -85,B 0,C 180,E1 -9022.577,E2 -9022.577} C_VEL
LIN {X 0,Y 439.397,Z 338.566,A -85,B 0,C 180,E1 -9025.586,E2 -9025.586} C_VEL
LIN {X 0,Y 439.417,Z 338.563,A -85,B 0,C 180,E1 -9028.674,E2 -9028.674} C_VEL
LIN {X 0,Y 439.366,Z 338.569,A -85,B 0,C 180,E1 -9031.862,E2 -9031.862} C_VEL
LIN {X 0,Y 439.394,Z 338.567,A -85,B 0,C 180,E1 -9035.157,E2 -9035.157} C_VEL
LIN {X 0,Y 439.382,Z 338.569,A -85,B 0,C 180,E1 -9038.596,E2 -9038.596} C_VEL
LIN {X 0,Y 439.383,Z 338.567,A -85,B 0,C 180,E1 -9041.258,E2 -9041.258} C_VEL
LIN {X 0,Y 439.4,Z 338.566,A -85,B 0,C 180,E1 -9044.73,E2 -9044.73} C_VEL
LIN {X 0,Y 439.393,Z 338.565,A -85,B 0,C 180,E1 -9047.797,E2 -9047.797} C_VEL
LIN {X 0,Y 439.432,Z 338.562,A -85,B 0,C 180,E1 -9050.23,E2 -9050.23} C_VEL
LIN {X 0,Y 439.431,Z 338.641,A -85,B 0,C 180,E1 -9052.956,E2 -9052.956} C_VEL
LIN {X 0,Y 440.398,Z 343.945,A -85,B 0,C 180,E1 -9055.495,E2 -9055.495} C_VEL
LIN {X 0,Y 440.722,Z 347.621,A -85,B 0,C 180,E1 -9057.169,E2 -9057.169} C_VEL
LIN {X 0,Y 440.254,Z 354.955,A -85,B 0,C 180,E1 -9060.341,E2 -9060.341} C_VEL
LIN {X 0,Y 439.715,Z 363.662,A -85,B 0,C 180,E1 -9063.967,E2 -9063.967} C_VEL
LIN {X 0,Y 439.326,Z 370.946,A -85,B 0,C 180,E1 -9066.927,E2 -9066.927} C_VEL
LIN {X 0,Y 438.998,Z 379.598,A -85,B 0,C 180,E1 -9070.356,E2 -9070.356} C_VEL
LIN {X 0,Y 438.718,Z 388.95,A -85,B 0,C 180,E1 -9073.981,E2 -9073.981} C_VEL
LIN {X 0,Y 438.51,Z 397.14,A -85,B 0,C 180,E1 -9077.114,E2 -9077.114} C_VEL
LIN {X 0,Y 439.93,Z 409.902,A -85,B 0,C 180,E1 -9077.6,E2 -9077.6} C_VEL
LIN {X 0,Y 440.542,Z 418.123,A -85,B 0,C 180,E1 -9078.032,E2 -9078.032} C_VEL
LIN {X 0,Y 440.182,Z 428.495,A -85,B 0,C 180,E1 -9078.722,E2 -9078.722} C_VEL
LIN {X 0,Y 439.828,Z 435.446,A -85,B 0,C 180,E1 -9079.296,E2 -9079.296} C_VEL
LIN {X 0,Y 439.445,Z 443.435,A -85,B 0,C 180,E1 -9080.102,E2 -9080.102} C_VEL
LIN {X 0,Y 439.195,Z 449.191,A -85,B 0,C 180,E1 -9080.793,E2 -9080.793} C_VEL
LIN {X 0,Y 438.917,Z 455.621,A -85,B 0,C 180,E1 -9081.716,E2 -9081.716} C_VEL
LIN {X 0,Y 438.702,Z 460.968,A -85,B 0,C 180,E1 -9082.638,E2 -9082.638} C_VEL
LIN {X 0,Y 438.505,Z 465.427,A -85,B 0,C 180,E1 -9083.56,E2 -9083.56} C_VEL
LIN {X 0,Y 438.439,Z 469.144,A -85,B 0,C 180,E1 -9084.482,E2 -9084.482} C_VEL
LIN {X 0,Y 438.367,Z 472.175,A -85,B 0,C 180,E1 -9085.403,E2 -9085.403} C_VEL
LIN {X 0,Y 438.341,Z 474.525,A -85,B 0,C 180,E1 -9086.324,E2 -9086.324} C_VEL
LIN {X 0,Y 438.386,Z 476.313,A -85,B 0,C 180,E1 -9087.245,E2 -9087.245} C_VEL
LIN {X 0,Y 438.319,Z 477.59,A -85,B 0,C 180,E1 -9088.164,E2 -9088.164} C_VEL
LIN {X 0,Y 438.304,Z 478.388,A -85,B 0,C 180,E1 -9089.082,E2 -9089.082} C_VEL
LIN {X 0,Y 438.308,Z 478.679,A -85,B 0,C 180,E1 -9090.001,E2 -9090.001} C_VEL
LIN {X 0,Y 438.304,Z 478.376,A -85,B 0,C 180,E1 -9090.92,E2 -9090.92} C_VEL
LIN {X 0,Y 438.319,Z 477.59,A -85,B 0,C 180,E1 -9091.839,E2 -9091.839} C_VEL
LIN {X 0,Y 438.386,Z 476.327,A -85,B 0,C 180,E1 -9092.758,E2 -9092.758} C_VEL
LIN {X 0,Y 438.325,Z 473.378,A -85,B 0,C 180,E1 -9094.139,E2 -9094.139} C_VEL
LIN {X 0,Y 438.446,Z 470.708,A -85,B 0,C 180,E1 -9095.059,E2 -9095.059} C_VEL
LIN {X 0,Y 438.457,Z 466.862,A -85,B 0,C 180,E1 -9096.111,E2 -9096.111} C_VEL
LIN {X 0,Y 438.667,Z 462.224,A -85,B 0,C 180,E1 -9097.134,E2 -9097.134} C_VEL
LIN {X 0,Y 438.837,Z 457.162,A -85,B 0,C 180,E1 -9098.057,E2 -9098.057} C_VEL
LIN {X 0,Y 439.118,Z 451.079,A -85,B 0,C 180,E1 -9098.979,E2 -9098.979} C_VEL
LIN {X 0,Y 439.48,Z 443.697,A -85,B 0,C 180,E1 -9099.9,E2 -9099.9} C_VEL
LIN {X 0,Y 439.841,Z 435.814,A -85,B 0,C 180,E1 -9100.706,E2 -9100.706} C_VEL
LIN {X 0,Y 440.265,Z 427.52,A -85,B 0,C 180,E1 -9101.394,E2 -9101.394} C_VEL
LIN {X 0,Y 440.578,Z 417.354,A -85,B 0,C 180,E1 -9102.065,E2 -9102.065} C_VEL
LIN {X 0,Y 439.587,Z 405.423,A -85,B 0,C 180,E1 -9102.656,E2 -9102.656} C_VEL
LIN {X 0,Y 438.512,Z 396.522,A -85,B 0,C 180,E1 -9102.997,E2 -9102.997} C_VEL
LIN {X 0,Y 438.692,Z 388.571,A -85,B 0,C 180,E1 -9106.008,E2 -9106.008} C_VEL
LIN {X 0,Y 438.921,Z 380.457,A -85,B 0,C 180,E1 -9109.142,E2 -9109.142} C_VEL
LIN {X 0,Y 439.162,Z 373.611,A -85,B 0,C 180,E1 -9111.846,E2 -9111.846} C_VEL
LIN {X 0,Y 439.621,Z 364.446,A -85,B 0,C 180,E1 -9115.572,E2 -9115.572} C_VEL
LIN {X 0,Y 440.066,Z 357.271,A -85,B 0,C 180,E1 -9118.628,E2 -9118.628} C_VEL
LIN {X 0,Y 440.601,Z 350.168,A -85,B 0,C 180,E1 -9121.762,E2 -9121.762} C_VEL
LIN {X 0,Y 440.706,Z 346.684,A -85,B 0,C 180,E1 -9123.38,E2 -9123.38} C_VEL
LIN {X 0,Y 439.802,Z 340.995,A -85,B 0,C 180,E1 -9126.247,E2 -9126.247} C_VEL
LIN {X 0,Y 439.379,Z 338.569,A -85,B 0,C 180,E1 -9127.578,E2 -9127.578} C_VEL
LIN {X 0,Y 439.412,Z 338.569,A -85,B 0,C 180,E1 -9129.85,E2 -9129.85} C_VEL
LIN {X 0,Y 439.388,Z 338.573,A -85,B 0,C 180,E1 -9132.627,E2 -9132.627} C_VEL
LIN {X 0,Y 439.406,Z 338.569,A -85,B 0,C 180,E1 -9135.271,E2 -9135.271} C_VEL
LIN {X 0,Y 439.395,Z 338.568,A -85,B 0,C 180,E1 -9138.744,E2 -9138.744} C_VEL
LIN {X 0,Y 439.376,Z 338.569,A -85,B 0,C 180,E1 -9141.609,E2 -9141.609} C_VEL
LIN {X 0,Y 439.403,Z 338.566,A -85,B 0,C 180,E1 -9144.844,E2 -9144.844} C_VEL
LIN {X 0,Y 439.378,Z 338.57,A -85,B 0,C 180,E1 -9148.139,E2 -9148.139} C_VEL
LIN {X 0,Y 439.44,Z 338.561,A -85,B 0,C 180,E1 -9151.598,E2 -9151.598} C_VEL
LIN {X 0,Y 439.408,Z 338.565,A -85,B 0,C 180,E1 -9154.415,E2 -9154.415} C_VEL
LIN {X 0,Y 439.372,Z 338.569,A -85,B 0,C 180,E1 -9157.424,E2 -9157.424} C_VEL
LIN {X 0,Y 439.448,Z 338.559,A -85,B 0,C 180,E1 -9160.663,E2 -9160.663} C_VEL
LIN {X 0,Y 439.469,Z 338.556,A -85,B 0,C 180,E1 -9164.224,E2 -9164.224} C_VEL
LIN {X 0,Y 439.49,Z 338.554,A -85,B 0,C 180,E1 -9168.001,E2 -9168.001} C_VEL
LIN {X 0,Y 439.51,Z 338.554,A -85,B 0,C 180,E1 -9171.725,E2 -9171.725} C_VEL
LIN {X 0,Y 439.615,Z 338.539,A -85,B 0,C 180,E1 -9174.495,E2 -9174.495} C_VEL
LIN {X 0,Y 439.639,Z 338.534,A -85,B 0,C 180,E1 -9178.167,E2 -9178.167} C_VEL
LIN {X 0,Y 439.768,Z 338.521,A -85,B 0,C 180,E1 -9179.999,E2 -9179.999} C_VEL
LIN {X 0,Y 439.644,Z 338.535,A -85,B 0,C 180,E1 -9182.748,E2 -9182.748} C_VEL
LIN {X 0,Y 439.612,Z 338.54,A -85,B 0,C 180,E1 -9186.424,E2 -9186.424} C_VEL
LIN {X 0,Y 439.499,Z 338.553,A -85,B 0,C 180,E1 -9189.201,E2 -9189.201} C_VEL
LIN {X 0,Y 439.47,Z 338.559,A -85,B 0,C 180,E1 -9192.936,E2 -9192.936} C_VEL
LIN {X 0,Y 439.448,Z 338.564,A -85,B 0,C 180,E1 -9196.346,E2 -9196.346} C_VEL
LIN {X 0,Y 439.134,Z 338.601,A -85,B 0,C 180,E1 -9199.22,E2 -9199.22} C_VEL
LIN {X 0,Y 439.033,Z 338.69,A -85,B 0,C 180,E1 -9199.642,E2 -9199.642} C_VEL
LIN {X 0,Y 438.914,Z 342.123,A -85,B 0,C 180,E1 -9202.599,E2 -9202.599} C_VEL
LIN {X 0,Y 438.859,Z 344.43,A -85,B 0,C 180,E1 -9204.604,E2 -9204.604} C_VEL
LIN {X 0,Y 438.727,Z 348.809,A -85,B 0,C 180,E1 -9208.229,E2 -9208.229} C_VEL
LIN {X 0,Y 438.616,Z 351.981,A -85,B 0,C 180,E1 -9210.845,E2 -9210.845} C_VEL
LIN {X 0,Y 438.531,Z 356.015,A -85,B 0,C 180,E1 -9214.118,E2 -9214.118} C_VEL
LIN {X 0,Y 438.434,Z 359.784,A -85,B 0,C 180,E1 -9217.135,E2 -9217.135} C_VEL
LIN {X 0,Y 440.676,Z 371.18,A -85,B 0,C 180,E1 -9217.661,E2 -9217.661} C_VEL
LIN {X 0,Y 441.202,Z 375.603,A -85,B 0,C 180,E1 -9217.897,E2 -9217.897} C_VEL
LIN {X 0,Y 440.775,Z 386.901,A -85,B 0,C 180,E1 -9218.62,E2 -9218.62} C_VEL
LIN {X 0,Y 440.343,Z 396.142,A -85,B 0,C 180,E1 -9219.398,E2 -9219.398} C_VEL
LIN {X 0,Y 439.97,Z 404.439,A -85,B 0,C 180,E1 -9220.273,E2 -9220.273} C_VEL
LIN {X 0,Y 439.563,Z 412.185,A -85,B 0,C 180,E1 -9221.281,E2 -9221.281} C_VEL
LIN {X 0,Y 439.231,Z 419.031,A -85,B 0,C 180,E1 -9222.407,E2 -9222.407} C_VEL
LIN {X 0,Y 438.902,Z 424.395,A -85,B 0,C 180,E1 -9223.513,E2 -9223.513} C_VEL
LIN {X 0,Y 438.769,Z 427.939,A -85,B 0,C 180,E1 -9224.394,E2 -9224.394} C_VEL
LIN {X 0,Y 438.559,Z 431.967,A -85,B 0,C 180,E1 -9225.7,E2 -9225.7} C_VEL
LIN {X 0,Y 438.439,Z 433.761,A -85,B 0,C 180,E1 -9226.426,E2 -9226.426} C_VEL
LIN {X 0,Y 438.324,Z 435.961,A -85,B 0,C 180,E1 -9227.667,E2 -9227.667} C_VEL
LIN {X 0,Y 438.27,Z 437.204,A -85,B 0,C 180,E1 -9228.908,E2 -9228.908} C_VEL
LIN {X 0,Y 438.214,Z 437.462,A -85,B 0,C 180,E1 -9230.335,E2 -9230.335} C_VEL
LIN {X 0,Y 438.248,Z 437.047,A -85,B 0,C 180,E1 -9231.285,E2 -9231.285} C_VEL
LIN {X 0,Y 438.313,Z 435.731,A -85,B 0,C 180,E1 -9232.46,E2 -9232.46} C_VEL
LIN {X 0,Y 438.445,Z 433.588,A -85,B 0,C 180,E1 -9233.623,E2 -9233.623} C_VEL
LIN {X 0,Y 438.564,Z 430.464,A -85,B 0,C 180,E1 -9234.811,E2 -9234.811} C_VEL
LIN {X 0,Y 438.787,Z 425.558,A -85,B 0,C 180,E1 -9236.176,E2 -9236.176} C_VEL
LIN {X 0,Y 439.025,Z 420.47,A -85,B 0,C 180,E1 -9237.281,E2 -9237.281} C_VEL
LIN {X 0,Y 439.3,Z 415.703,A -85,B 0,C 180,E1 -9238.133,E2 -9238.133} C_VEL
LIN {X 0,Y 439.608,Z 409.224,A -85,B 0,C 180,E1 -9239.096,E2 -9239.096} C_VEL
LIN {X 0,Y 439.917,Z 402.01,A -85,B 0,C 180,E1 -9239.979,E2 -9239.979} C_VEL
LIN {X 0,Y 440.3,Z 393.097,A -85,B 0,C 180,E1 -9240.867,E2 -9240.867} C_VEL
LIN {X 0,Y 440.733,Z 382.413,A -85,B 0,C 180,E1 -9241.679,E2 -9241.679} C_VEL
LIN {X 0,Y 440.924,Z 373.248,A -85,B 0,C 180,E1 -9242.21,E2 -9242.21} C_VEL
LIN {X 0,Y 439.249,Z 363.614,A -85,B 0,C 180,E1 -9242.676,E2 -9242.676} C_VEL
LIN {X 0,Y 438.475,Z 359.142,A -85,B 0,C 180,E1 -9242.882,E2 -9242.882} C_VEL
LIN {X 0,Y 438.488,Z 354.629,A -85,B 0,C 180,E1 -9246.377,E2 -9246.377} C_VEL
LIN {X 0,Y 438.513,Z 350.825,A -85,B 0,C 180,E1 -9249.353,E2 -9249.353} C_VEL
LIN {X 0,Y 438.627,Z 347.163,A -85,B 0,C 180,E1 -9252.275,E2 -9252.275} C_VEL
LIN {X 0,Y 438.712,Z 343.582,A -85,B 0,C 180,E1 -9255.147,E2 -9255.147} C_VEL
LIN {X 0,Y 438.879,Z 340.113,A -85,B 0,C 180,E1 -9257.983,E2 -9257.983} C_VEL
LIN {X 0,Y 438.924,Z 338.969,A -85,B 0,C 180,E1 -9258.921,E2 -9258.921} C_VEL
LIN {X 0,Y 439.127,Z 338.599,A -85,B 0,C 180,E1 -9260.516,E2 -9260.516} C_VEL
LIN {X 0,Y 438.647,Z 338.662,A -85,B 0,C 180,E1 -9261.282,E2 -9261.282} C_VEL
LIN {X 0,Y 436.074,Z 338.986,A -85,B 0,C 180,E1 -9262.533,E2 -9262.533} C_VEL
LIN {X 0,Y 432.932,Z 339.374,A -85,B 0,C 180,E1 -9264.057,E2 -9264.057} C_VEL
LIN {X 0,Y 432.535,Z 339.42,A -85,B 0,C 180,E1 -9264.582,E2 -9264.582} C_VEL
LIN {X 0,Y 432.596,Z 339.414,A -85,B 0,C 180,E1 -9268.137,E2 -9268.137} C_VEL
LIN {X 0,Y 432.723,Z 339.398,A -85,B 0,C 180,E1 -9269.999,E2 -9269.999} C_VEL
LIN {X 0,Y 432.596,Z 339.412,A -85,B 0,C 180,E1 -9272.792,E2 -9272.792} C_VEL
LIN {X 0,Y 432.565,Z 339.417,A -85,B 0,C 180,E1 -9276.529,E2 -9276.529} C_VEL
LIN {X 0,Y 432.434,Z 339.432,A -85,B 0,C 180,E1 -9279.352,E2 -9279.352} C_VEL
LIN {X 0,Y 432.432,Z 339.432,A -85,B 0,C 180,E1 -9282.811,E2 -9282.811} C_VEL
LIN {X 0,Y 432.399,Z 339.436,A -85,B 0,C 180,E1 -9286.478,E2 -9286.478} C_VEL
LIN {X 0,Y 432.326,Z 339.448,A -85,B 0,C 180,E1 -9289.96,E2 -9289.96} C_VEL
LIN {X 0,Y 432.305,Z 339.449,A -85,B 0,C 180,E1 -9292.963,E2 -9292.963} C_VEL
LIN {X 0,Y 432.351,Z 339.444,A -85,B 0,C 180,E1 -9296.032,E2 -9296.032} C_VEL
LIN {X 0,Y 432.338,Z 339.446,A -85,B 0,C 180,E1 -9299.186,E2 -9299.186} C_VEL
LIN {X 0,Y 432.311,Z 339.447,A -85,B 0,C 180,E1 -9302.293,E2 -9302.293} C_VEL
LIN {X 0,Y 432.326,Z 339.445,A -85,B 0,C 180,E1 -9304.676,E2 -9304.676} C_VEL
LIN {X 0,Y 432.339,Z 339.443,A -85,B 0,C 180,E1 -9308.148,E2 -9308.148} C_VEL
LIN {X 0,Y 432.358,Z 339.443,A -85,B 0,C 180,E1 -9311.608,E2 -9311.608} C_VEL
LIN {X 0,Y 432.363,Z 339.44,A -85,B 0,C 180,E1 -9314.341,E2 -9314.341} C_VEL
LIN {X 0,Y 432.351,Z 339.445,A -85,B 0,C 180,E1 -9317.009,E2 -9317.009} C_VEL
LIN {X 0,Y 432.343,Z 339.442,A -85,B 0,C 180,E1 -9319.817,E2 -9319.817} C_VEL
LIN {X 0,Y 432.303,Z 339.451,A -85,B 0,C 180,E1 -9323.023,E2 -9323.023} C_VEL
LIN {X 0,Y 432.345,Z 339.443,A -85,B 0,C 180,E1 -9325.997,E2 -9325.997} C_VEL
LIN {X 0,Y 432.38,Z 339.437,A -85,B 0,C 180,E1 -9329.744,E2 -9329.744} C_VEL
LIN {X 0,Y 432.385,Z 339.437,A -85,B 0,C 180,E1 -9333.373,E2 -9333.373} C_VEL
LIN {X 0,Y 432.36,Z 339.441,A -85,B 0,C 180,E1 -9336.024,E2 -9336.024} C_VEL
LIN {X 0,Y 432.355,Z 339.441,A -85,B 0,C 180,E1 -9339.048,E2 -9339.048} C_VEL
LIN {X 0,Y 432.365,Z 339.441,A -85,B 0,C 180,E1 -9342.012,E2 -9342.012} C_VEL
LIN {X 0,Y 432.388,Z 339.438,A -85,B 0,C 180,E1 -9344.927,E2 -9344.927} C_VEL
LIN {X 0,Y 432.468,Z 339.429,A -85,B 0,C 180,E1 -9347.805,E2 -9347.805} C_VEL
LIN {X 0,Y 432.48,Z 339.427,A -85,B 0,C 180,E1 -9351.591,E2 -9351.591} C_VEL
LIN {X 0,Y 432.587,Z 339.415,A -85,B 0,C 180,E1 -9354.407,E2 -9354.407} C_VEL
LIN {X 0,Y 432.594,Z 339.415,A -85,B 0,C 180,E1 -9358.139,E2 -9358.139} C_VEL
LIN {X 0,Y 432.722,Z 339.398,A -85,B 0,C 180,E1 -9360.001,E2 -9360.001} C_VEL
LIN {X 0,Y 432.597,Z 339.411,A -85,B 0,C 180,E1 -9362.794,E2 -9362.794} C_VEL
LIN {X 0,Y 432.562,Z 339.416,A -85,B 0,C 180,E1 -9366.531,E2 -9366.531} C_VEL
LIN {X 0,Y 432.435,Z 339.434,A -85,B 0,C 180,E1 -9369.354,E2 -9369.354} C_VEL
LIN {X 0,Y 432.435,Z 339.432,A -85,B 0,C 180,E1 -9372.813,E2 -9372.813} C_VEL
LIN {X 0,Y 432.403,Z 339.435,A -85,B 0,C 180,E1 -9376.48,E2 -9376.48} C_VEL
LIN {X 0,Y 432.329,Z 339.446,A -85,B 0,C 180,E1 -9379.962,E2 -9379.962} C_VEL
LIN {X 0,Y 432.311,Z 339.449,A -85,B 0,C 180,E1 -9382.965,E2 -9382.965} C_VEL
LIN {X 0,Y 432.356,Z 339.442,A -85,B 0,C 180,E1 -9386.034,E2 -9386.034} C_VEL
LIN {X 0,Y 432.345,Z 339.445,A -85,B 0,C 180,E1 -9389.188,E2 -9389.188} C_VEL
LIN {X 0,Y 432.318,Z 339.446,A -85,B 0,C 180,E1 -9392.295,E2 -9392.295} C_VEL
LIN {X 0,Y 432.334,Z 339.445,A -85,B 0,C 180,E1 -9394.678,E2 -9394.678} C_VEL
LIN {X 0,Y 432.34,Z 339.443,A -85,B 0,C 180,E1 -9398.15,E2 -9398.15} C_VEL
LIN {X 0,Y 432.328,Z 339.446,A -85,B 0,C 180,E1 -9401.604,E2 -9401.604} C_VEL
LIN {X 0,Y 432.335,Z 339.445,A -85,B 0,C 180,E1 -9404.348,E2 -9404.348} C_VEL
LIN {X 0,Y 432.32,Z 339.448,A -85,B 0,C 180,E1 -9407.016,E2 -9407.016} C_VEL
LIN {X 0,Y 432.337,Z 339.445,A -85,B 0,C 180,E1 -9409.821,E2 -9409.821} C_VEL
LIN {X 0,Y 432.404,Z 339.579,A -85,B 0,C 180,E1 -9412.789,E2 -9412.789} C_VEL
LIN {X 0,Y 433.494,Z 345.729,A -85,B 0,C 180,E1 -9415.776,E2 -9415.776} C_VEL
LIN {X 0,Y 433.683,Z 349.871,A -85,B 0,C 180,E1 -9417.673,E2 -9417.673} C_VEL
LIN {X 0,Y 433.063,Z 357.975,A -85,B 0,C 180,E1 -9421.205,E2 -9421.205} C_VEL
LIN {X 0,Y 432.586,Z 365.781,A -85,B 0,C 180,E1 -9424.5,E2 -9424.5} C_VEL
LIN {X 0,Y 432.184,Z 373.177,A -85,B 0,C 180,E1 -9427.535,E2 -9427.535} C_VEL
LIN {X 0,Y 431.868,Z 381.057,A -85,B 0,C 180,E1 -9430.711,E2 -9430.711} C_VEL
LIN {X 0,Y 431.644,Z 389.198,A -85,B 0,C 180,E1 -9433.933,E2 -9433.933} C_VEL
LIN {X 0,Y 431.444,Z 396.862,A -85,B 0,C 180,E1 -9436.914,E2 -9436.914} C_VEL
LIN {X 0,Y 432.814,Z 409.346,A -85,B 0,C 180,E1 -9437.395,E2 -9437.395} C_VEL
LIN {X 0,Y 433.516,Z 419.47,A -85,B 0,C 180,E1 -9437.954,E2 -9437.954} C_VEL
LIN {X 0,Y 433.207,Z 428.017,A -85,B 0,C 180,E1 -9438.538,E2 -9438.538} C_VEL
LIN {X 0,Y 432.774,Z 436.227,A -85,B 0,C 180,E1 -9439.238,E2 -9439.238} C_VEL
LIN {X 0,Y 432.381,Z 444.032,A -85,B 0,C 180,E1 -9440.056,E2 -9440.056} C_VEL
LIN {X 0,Y 432.093,Z 450.496,A -85,B 0,C 180,E1 -9440.877,E2 -9440.877} C_VEL
LIN {X 0,Y 431.786,Z 456.655,A -85,B 0,C 180,E1 -9441.813,E2 -9441.813} C_VEL
LIN {X 0,Y 431.528,Z 462.948,A -85,B 0,C 180,E1 -9442.985,E2 -9442.985} C_VEL
LIN {X 0,Y 431.341,Z 468.783,A -85,B 0,C 180,E1 -9444.391,E2 -9444.391} C_VEL
LIN {X 0,Y 431.3,Z 471.819,A -85,B 0,C 180,E1 -9445.328,E2 -9445.328} C_VEL
LIN {X 0,Y 431.241,Z 474.172,A -85,B 0,C 180,E1 -9446.264,E2 -9446.264} C_VEL
LIN {X 0,Y 431.296,Z 475.966,A -85,B 0,C 180,E1 -9447.199,E2 -9447.199} C_VEL
LIN {X 0,Y 431.242,Z 477.25,A -85,B 0,C 180,E1 -9448.133,E2 -9448.133} C_VEL
LIN {X 0,Y 431.218,Z 478.053,A -85,B 0,C 180,E1 -9449.067,E2 -9449.067} C_VEL
LIN {X 0,Y 431.22,Z 478.345,A -85,B 0,C 180,E1 -9450.001,E2 -9450.001} C_VEL
LIN {X 0,Y 431.218,Z 478.044,A -85,B 0,C 180,E1 -9450.935,E2 -9450.935} C_VEL
LIN {X 0,Y 431.242,Z 477.262,A -85,B 0,C 180,E1 -9451.869,E2 -9451.869} C_VEL
LIN {X 0,Y 431.296,Z 476.002,A -85,B 0,C 180,E1 -9452.803,E2 -9452.803} C_VEL
LIN {X 0,Y 431.243,Z 473.06,A -85,B 0,C 180,E1 -9454.207,E2 -9454.207} C_VEL
LIN {X 0,Y 431.354,Z 470.395,A -85,B 0,C 180,E1 -9455.142,E2 -9455.142} C_VEL
LIN {X 0,Y 431.444,Z 465.164,A -85,B 0,C 180,E1 -9456.549,E2 -9456.549} C_VEL
LIN {X 0,Y 431.692,Z 459.555,A -85,B 0,C 180,E1 -9457.72,E2 -9457.72} C_VEL
LIN {X 0,Y 431.992,Z 452.522,A -85,B 0,C 180,E1 -9458.892,E2 -9458.892} C_VEL
LIN {X 0,Y 432.413,Z 444.479,A -85,B 0,C 180,E1 -9459.945,E2 -9459.945} C_VEL
LIN {X 0,Y 432.817,Z 436.825,A -85,B 0,C 180,E1 -9460.763,E2 -9460.763} C_VEL
LIN {X 0,Y 433.23,Z 428.823,A -85,B 0,C 180,E1 -9461.463,E2 -9461.463} C_VEL
LIN {X 0,Y 433.584,Z 420.587,A -85,B 0,C 180,E1 -9462.047,E2 -9462.047} C_VEL
LIN {X 0,Y 433.16,Z 412.377,A -85,B 0,C 180,E1 -9462.529,E2 -9462.529} C_VEL
LIN {X 0,Y 432.263,Z 403.017,A -85,B 0,C 180,E1 -9462.962,E2 -9462.962} C_VEL
LIN {X 0,Y 431.42,Z 396.218,A -85,B 0,C 180,E1 -9463.214,E2 -9463.214} C_VEL
LIN {X 0,Y 431.668,Z 387.715,A -85,B 0,C 180,E1 -9466.506,E2 -9466.506} C_VEL
LIN {X 0,Y 431.946,Z 378.947,A -85,B 0,C 180,E1 -9469.98,E2 -9469.98} C_VEL
LIN {X 0,Y 432.281,Z 370.369,A -85,B 0,C 180,E1 -9473.474,E2 -9473.474} C_VEL
LIN {X 0,Y 432.722,Z 362.694,A -85,B 0,C 180,E1 -9476.711,E2 -9476.711} C_VEL
LIN {X 0,Y 433.318,Z 354.798,A -85,B 0,C 180,E1 -9480.186,E2 -9480.186} C_VEL
LIN {X 0,Y 433.769,Z 349.543,A -85,B 0,C 180,E1 -9482.593,E2 -9482.593} C_VEL
LIN {X 0,Y 433.401,Z 345.517,A -85,B 0,C 180,E1 -9484.581,E2 -9484.581} C_VEL
LIN {X 0,Y 432.358,Z 339.444,A -85,B 0,C 180,E1 -9487.897,E2 -9487.897} C_VEL
LIN {X 0,Y 432.332,Z 339.453,A -85,B 0,C 180,E1 -9490.561,E2 -9490.561} C_VEL
LIN {X 0,Y 432.324,Z 339.454,A -85,B 0,C 180,E1 -9493.061,E2 -9493.061} C_VEL
LIN {X 0,Y 432.34,Z 339.448,A -85,B 0,C 180,E1 -9495.665,E2 -9495.665} C_VEL
LIN {X 0,Y 432.339,Z 339.446,A -85,B 0,C 180,E1 -9498.398,E2 -9498.398} C_VEL
LIN {X 0,Y 432.34,Z 339.445,A -85,B 0,C 180,E1 -9501.85,E2 -9501.85} C_VEL
LIN {X 0,Y 432.344,Z 339.444,A -85,B 0,C 180,E1 -9505.323,E2 -9505.323} C_VEL
LIN {X 0,Y 432.327,Z 339.446,A -85,B 0,C 180,E1 -9508.654,E2 -9508.654} C_VEL
LIN {X 0,Y 432.389,Z 339.44,A -85,B 0,C 180,E1 -9511.877,E2 -9511.877} C_VEL
LIN {X 0,Y 432.356,Z 339.443,A -85,B 0,C 180,E1 -9514.998,E2 -9514.998} C_VEL
LIN {X 0,Y 432.365,Z 339.441,A -85,B 0,C 180,E1 -9518.045,E2 -9518.045} C_VEL
LIN {X 0,Y 432.391,Z 339.44,A -85,B 0,C 180,E1 -9521.029,E2 -9521.029} C_VEL
LIN {X 0,Y 432.437,Z 339.432,A -85,B 0,C 180,E1 -9523.961,E2 -9523.961} C_VEL
LIN {X 0,Y 432.466,Z 339.428,A -85,B 0,C 180,E1 -9527.803,E2 -9527.803} C_VEL
LIN {X 0,Y 432.47,Z 339.429,A -85,B 0,C 180,E1 -9531.589,E2 -9531.589} C_VEL
LIN {X 0,Y 432.59,Z 339.414,A -85,B 0,C 180,E1 -9534.405,E2 -9534.405} C_VEL
LIN {X 0,Y 432.608,Z 339.41,A -85,B 0,C 180,E1 -9538.137,E2 -9538.137} C_VEL
LIN {X 0,Y 432.737,Z 339.397,A -85,B 0,C 180,E1 -9539.999,E2 -9539.999} C_VEL
LIN {X 0,Y 432.595,Z 339.412,A -85,B 0,C 180,E1 -9542.793,E2 -9542.793} C_VEL
LIN {X 0,Y 432.598,Z 339.412,A -85,B 0,C 180,E1 -9545.593,E2 -9545.593} C_VEL
LIN {X 0,Y 432.468,Z 339.43,A -85,B 0,C 180,E1 -9548.409,E2 -9548.409} C_VEL
LIN {X 0,Y 432.463,Z 339.431,A -85,B 0,C 180,E1 -9552.195,E2 -9552.195} C_VEL
LIN {X 0,Y 432.431,Z 339.437,A -85,B 0,C 180,E1 -9556.038,E2 -9556.038} C_VEL
LIN {X 0,Y 432.072,Z 339.481,A -85,B 0,C 180,E1 -9559.365,E2 -9559.365} C_VEL
LIN {X 0,Y 431.89,Z 342.226,A -85,B 0,C 180,E1 -9561.978,E2 -9561.978} C_VEL
LIN {X 0,Y 431.769,Z 345.784,A -85,B 0,C 180,E1 -9565.036,E2 -9565.036} C_VEL
LIN {X 0,Y 431.662,Z 349.82,A -85,B 0,C 180,E1 -9568.454,E2 -9568.454} C_VEL
LIN {X 0,Y 431.514,Z 353.375,A -85,B 0,C 180,E1 -9571.41,E2 -9571.41} C_VEL
LIN {X 0,Y 431.417,Z 357.491,A -85,B 0,C 180,E1 -9574.76,E2 -9574.76} C_VEL
LIN {X 0,Y 431.385,Z 360.224,A -85,B 0,C 180,E1 -9576.91,E2 -9576.91} C_VEL
LIN {X 0,Y 433.645,Z 371.591,A -85,B 0,C 180,E1 -9577.448,E2 -9577.448} C_VEL
LIN {X 0,Y 434.284,Z 376.26,A -85,B 0,C 180,E1 -9577.705,E2 -9577.705} C_VEL
LIN {X 0,Y 433.858,Z 387.369,A -85,B 0,C 180,E1 -9578.434,E2 -9578.434} C_VEL
LIN {X 0,Y 433.47,Z 395.586,A -85,B 0,C 180,E1 -9579.128,E2 -9579.128} C_VEL
LIN {X 0,Y 433.086,Z 402.731,A -85,B 0,C 180,E1 -9579.864,E2 -9579.864} C_VEL
LIN {X 0,Y 432.695,Z 410.044,A -85,B 0,C 180,E1 -9580.782,E2 -9580.782} C_VEL
LIN {X 0,Y 432.371,Z 416.615,A -85,B 0,C 180,E1 -9581.791,E2 -9581.791} C_VEL
LIN {X 0,Y 431.951,Z 423.508,A -85,B 0,C 180,E1 -9583.105,E2 -9583.105} C_VEL
LIN {X 0,Y 431.683,Z 428.737,A -85,B 0,C 180,E1 -9584.43,E2 -9584.43} C_VEL
LIN {X 0,Y 431.461,Z 432.708,A -85,B 0,C 180,E1 -9585.781,E2 -9585.781} C_VEL
LIN {X 0,Y 431.279,Z 435.55,A -85,B 0,C 180,E1 -9587.162,E2 -9587.162} C_VEL
LIN {X 0,Y 431.178,Z 437.285,A -85,B 0,C 180,E1 -9588.569,E2 -9588.569} C_VEL
LIN {X 0,Y 431.12,Z 437.887,A -85,B 0,C 180,E1 -9590.01,E2 -9590.01} C_VEL
LIN {X 0,Y 431.158,Z 436.932,A -85,B 0,C 180,E1 -9591.726,E2 -9591.726} C_VEL
LIN {X 0,Y 431.369,Z 434.198,A -85,B 0,C 180,E1 -9593.542,E2 -9593.542} C_VEL
LIN {X 0,Y 431.5,Z 430.736,A -85,B 0,C 180,E1 -9594.893,E2 -9594.893} C_VEL
LIN {X 0,Y 431.699,Z 426.455,A -85,B 0,C 180,E1 -9596.124,E2 -9596.124} C_VEL
LIN {X 0,Y 431.946,Z 421.49,A -85,B 0,C 180,E1 -9597.247,E2 -9597.247} C_VEL
LIN {X 0,Y 432.305,Z 415.252,A -85,B 0,C 180,E1 -9598.378,E2 -9598.378} C_VEL
LIN {X 0,Y 432.666,Z 408.192,A -85,B 0,C 180,E1 -9599.415,E2 -9599.415} C_VEL
LIN {X 0,Y 433.068,Z 399.298,A -85,B 0,C 180,E1 -9600.465,E2 -9600.465} C_VEL
LIN {X 0,Y 433.507,Z 389.904,A -85,B 0,C 180,E1 -9601.319,E2 -9601.319} C_VEL
LIN {X 0,Y 433.811,Z 381.798,A -85,B 0,C 180,E1 -9601.911,E2 -9601.911} C_VEL
LIN {X 0,Y 433.935,Z 373.851,A -85,B 0,C 180,E1 -9602.379,E2 -9602.379} C_VEL
LIN {X 0,Y 432.27,Z 364.326,A -85,B 0,C 180,E1 -9602.854,E2 -9602.854} C_VEL
LIN {X 0,Y 431.395,Z 359.451,A -85,B 0,C 180,E1 -9603.077,E2 -9603.077} C_VEL
LIN {X 0,Y 431.402,Z 355.744,A -85,B 0,C 180,E1 -9605.965,E2 -9605.965} C_VEL
LIN {X 0,Y 431.441,Z 351.912,A -85,B 0,C 180,E1 -9608.999,E2 -9608.999} C_VEL
LIN {X 0,Y 431.544,Z 348.19,A -85,B 0,C 180,E1 -9611.974,E2 -9611.974} C_VEL
LIN {X 0,Y 431.663,Z 344.584,A -85,B 0,C 180,E1 -9614.899,E2 -9614.899} C_VEL
LIN {X 0,Y 431.827,Z 341.079,A -85,B 0,C 180,E1 -9617.784,E2 -9617.784} C_VEL
LIN {X 0,Y 431.845,Z 339.936,A -85,B 0,C 180,E1 -9618.737,E2 -9618.737} C_VEL
LIN {X 0,Y 431.957,Z 339.494,A -85,B 0,C 180,E1 -9619.689,E2 -9619.689} C_VEL
LIN {X 0,Y 432.456,Z 339.431,A -85,B 0,C 180,E1 -9622.529,E2 -9622.529} C_VEL
LIN {X 0,Y 432.535,Z 339.42,A -85,B 0,C 180,E1 -9624.582,E2 -9624.582} C_VEL
LIN {X 0,Y 431.758,Z 339.515,A -85,B 0,C 180,E1 -9625.359,E2 -9625.359} C_VEL
LIN {X 0,Y 428.922,Z 339.871,A -85,B 0,C 180,E1 -9626.624,E2 -9626.624} C_VEL
LIN {X 0,Y 426.601,Z 340.16,A -85,B 0,C 180,E1 -9627.645,E2 -9627.645} C_VEL
LIN {X 0,Y 425.617,Z 340.283,A -85,B 0,C 180,E1 -9628.433,E2 -9628.433} C_VEL
LIN {X 0,Y 425.538,Z 340.289,A -85,B 0,C 180,E1 -9628.699,E2 -9628.699} C_VEL
LIN {X 0,Y 425.692,Z 340.274,A -85,B 0,C 180,E1 -9629.999,E2 -9629.999} C_VEL
LIN {X 0,Y 425.548,Z 340.289,A -85,B 0,C 180,E1 -9632.839,E2 -9632.839} C_VEL
LIN {X 0,Y 425.567,Z 340.289,A -85,B 0,C 180,E1 -9635.685,E2 -9635.685} C_VEL
LIN {X 0,Y 425.431,Z 340.304,A -85,B 0,C 180,E1 -9638.549,E2 -9638.549} C_VEL
LIN {X 0,Y 425.418,Z 340.307,A -85,B 0,C 180,E1 -9642.4,E2 -9642.4} C_VEL
LIN {X 0,Y 425.375,Z 340.312,A -85,B 0,C 180,E1 -9646.311,E2 -9646.311} C_VEL
LIN {X 0,Y 425.315,Z 340.32,A -85,B 0,C 180,E1 -9649.635,E2 -9649.635} C_VEL
LIN {X 0,Y 425.293,Z 340.323,A -85,B 0,C 180,E1 -9653.364,E2 -9653.364} C_VEL
LIN {X 0,Y 425.335,Z 340.317,A -85,B 0,C 180,E1 -9656.844,E2 -9656.844} C_VEL
LIN {X 0,Y 425.304,Z 340.322,A -85,B 0,C 180,E1 -9659.717,E2 -9659.717} C_VEL
LIN {X 0,Y 425.268,Z 340.326,A -85,B 0,C 180,E1 -9663.047,E2 -9663.047} C_VEL
LIN {X 0,Y 425.27,Z 340.324,A -85,B 0,C 180,E1 -9665.929,E2 -9665.929} C_VEL
LIN {X 0,Y 425.299,Z 340.322,A -85,B 0,C 180,E1 -9669.046,E2 -9669.046} C_VEL
LIN {X 0,Y 425.317,Z 340.32,A -85,B 0,C 180,E1 -9672.646,E2 -9672.646} C_VEL
LIN {X 0,Y 425.304,Z 340.319,A -85,B 0,C 180,E1 -9676.052,E2 -9676.052} C_VEL
LIN {X 0,Y 425.295,Z 340.323,A -85,B 0,C 180,E1 -9678.626,E2 -9678.626} C_VEL
LIN {X 0,Y 425.31,Z 340.321,A -85,B 0,C 180,E1 -9681.104,E2 -9681.104} C_VEL
LIN {X 0,Y 425.286,Z 340.324,A -85,B 0,C 180,E1 -9684.664,E2 -9684.664} C_VEL
LIN {X 0,Y 425.257,Z 340.326,A -85,B 0,C 180,E1 -9688.074,E2 -9688.074} C_VEL
LIN {X 0,Y 425.323,Z 340.318,A -85,B 0,C 180,E1 -9691.369,E2 -9691.369} C_VEL
LIN {X 0,Y 425.282,Z 340.325,A -85,B 0,C 180,E1 -9694.555,E2 -9694.555} C_VEL
LIN {X 0,Y 425.312,Z 340.319,A -85,B 0,C 180,E1 -9697.719,E2 -9697.719} C_VEL
LIN {X 0,Y 425.352,Z 340.316,A -85,B 0,C 180,E1 -9700.705,E2 -9700.705} C_VEL
LIN {X 0,Y 425.385,Z 340.31,A -85,B 0,C 180,E1 -9703.689,E2 -9703.689} C_VEL
LIN {X 0,Y 425.417,Z 340.306,A -85,B 0,C 180,E1 -9707.599,E2 -9707.599} C_VEL
LIN {X 0,Y 425.43,Z 340.304,A -85,B 0,C 180,E1 -9711.451,E2 -9711.451} C_VEL
LIN {X 0,Y 425.543,Z 340.293,A -85,B 0,C 180,E1 -9714.314,E2 -9714.314} C_VEL
LIN {X 0,Y 425.564,Z 340.291,A -85,B 0,C 180,E1 -9718.108,E2 -9718.108} C_VEL
LIN {X 0,Y 425.691,Z 340.274,A -85,B 0,C 180,E1 -9720.001,E2 -9720.001} C_VEL
LIN {X 0,Y 425.549,Z 340.289,A -85,B 0,C 180,E1 -9722.841,E2 -9722.841} C_VEL
LIN {X 0,Y 425.52,Z 340.293,A -85,B 0,C 180,E1 -9726.64,E2 -9726.64} C_VEL
LIN {X 0,Y 425.394,Z 340.311,A -85,B 0,C 180,E1 -9729.51,E2 -9729.51} C_VEL
LIN {X 0,Y 425.394,Z 340.309,A -85,B 0,C 180,E1 -9732.911,E2 -9732.911} C_VEL
LIN {X 0,Y 425.352,Z 340.314,A -85,B 0,C 180,E1 -9736.606,E2 -9736.606} C_VEL
LIN {X 0,Y 425.319,Z 340.32,A -85,B 0,C 180,E1 -9739.637,E2 -9739.637} C_VEL
LIN {X 0,Y 425.298,Z 340.323,A -85,B 0,C 180,E1 -9743.366,E2 -9743.366} C_VEL
LIN {X 0,Y 425.341,Z 340.316,A -85,B 0,C 180,E1 -9746.846,E2 -9746.846} C_VEL
LIN {X 0,Y 425.31,Z 340.32,A -85,B 0,C 180,E1 -9749.719,E2 -9749.719} C_VEL
LIN {X 0,Y 425.275,Z 340.325,A -85,B 0,C 180,E1 -9753.049,E2 -9753.049} C_VEL
LIN {X 0,Y 425.278,Z 340.323,A -85,B 0,C 180,E1 -9755.931,E2 -9755.931} C_VEL
LIN {X 0,Y 425.294,Z 340.323,A -85,B 0,C 180,E1 -9759.045,E2 -9759.045} C_VEL
LIN {X 0,Y 425.272,Z 340.325,A -85,B 0,C 180,E1 -9762.654,E2 -9762.654} C_VEL
LIN {X 0,Y 425.263,Z 340.325,A -85,B 0,C 180,E1 -9766.046,E2 -9766.046} C_VEL
LIN {X 0,Y 425.28,Z 340.324,A -85,B 0,C 180,E1 -9769.48,E2 -9769.48} C_VEL
LIN {X 0,Y 425.322,Z 340.425,A -85,B 0,C 180,E1 -9772.566,E2 -9772.566} C_VEL
LIN {X 0,Y 426.531,Z 347.234,A -85,B 0,C 180,E1 -9775.931,E2 -9775.931} C_VEL
LIN {X 0,Y 426.666,Z 350.977,A -85,B 0,C 180,E1 -9777.671,E2 -9777.671} C_VEL
LIN {X 0,Y 425.98,Z 359.44,A -85,B 0,C 180,E1 -9781.417,E2 -9781.417} C_VEL
LIN {X 0,Y 425.538,Z 366.77,A -85,B 0,C 180,E1 -9784.572,E2 -9784.572} C_VEL
LIN {X 0,Y 425.091,Z 374.487,A -85,B 0,C 180,E1 -9787.797,E2 -9787.797} C_VEL
LIN {X 0,Y 424.769,Z 382.744,A -85,B 0,C 180,E1 -9791.179,E2 -9791.179} C_VEL
LIN {X 0,Y 424.539,Z 390.247,A -85,B 0,C 180,E1 -9794.203,E2 -9794.203} C_VEL
LIN {X 0,Y 424.347,Z 396.532,A -85,B 0,C 180,E1 -9796.699,E2 -9796.699} C_VEL
LIN {X 0,Y 425.753,Z 409.25,A -85,B 0,C 180,E1 -9797.211,E2 -9797.211} C_VEL
LIN {X 0,Y 426.484,Z 418.885,A -85,B 0,C 180,E1 -9797.752,E2 -9797.752} C_VEL
LIN {X 0,Y 426.221,Z 427.484,A -85,B 0,C 180,E1 -9798.348,E2 -9798.348} C_VEL
LIN {X 0,Y 425.778,Z 435.73,A -85,B 0,C 180,E1 -9799.059,E2 -9799.059} C_VEL
LIN {X 0,Y 425.364,Z 443.563,A -85,B 0,C 180,E1 -9799.891,E2 -9799.891} C_VEL
LIN {X 0,Y 425.033,Z 450.047,A -85,B 0,C 180,E1 -9800.724,E2 -9800.724} C_VEL
LIN {X 0,Y 424.752,Z 456.229,A -85,B 0,C 180,E1 -9801.677,E2 -9801.677} C_VEL
LIN {X 0,Y 424.45,Z 462.538,A -85,B 0,C 180,E1 -9802.868,E2 -9802.868} C_VEL
LIN {X 0,Y 424.249,Z 468.403,A -85,B 0,C 180,E1 -9804.297,E2 -9804.297} C_VEL
LIN {X 0,Y 424.232,Z 471.446,A -85,B 0,C 180,E1 -9805.25,E2 -9805.25} C_VEL
LIN {X 0,Y 424.147,Z 473.805,A -85,B 0,C 180,E1 -9806.201,E2 -9806.201} C_VEL
LIN {X 0,Y 424.208,Z 475.611,A -85,B 0,C 180,E1 -9807.152,E2 -9807.152} C_VEL
LIN {X 0,Y 424.167,Z 476.904,A -85,B 0,C 180,E1 -9808.102,E2 -9808.102} C_VEL
LIN {X 0,Y 424.135,Z 477.715,A -85,B 0,C 180,E1 -9809.052,E2 -9809.052} C_VEL
LIN {X 0,Y 424.134,Z 478.01,A -85,B 0,C 180,E1 -9810.001,E2 -9810.001} C_VEL
LIN {X 0,Y 424.135,Z 477.714,A -85,B 0,C 180,E1 -9810.951,E2 -9810.951} C_VEL
LIN {X 0,Y 424.167,Z 476.942,A -85,B 0,C 180,E1 -9811.9,E2 -9811.9} C_VEL
LIN {X 0,Y 424.193,Z 475.688,A -85,B 0,C 180,E1 -9812.85,E2 -9812.85} C_VEL
LIN {X 0,Y 424.165,Z 472.754,A -85,B 0,C 180,E1 -9814.277,E2 -9814.277} C_VEL
LIN {X 0,Y 424.265,Z 470.096,A -85,B 0,C 180,E1 -9815.229,E2 -9815.229} C_VEL
LIN {X 0,Y 424.337,Z 465.872,A -85,B 0,C 180,E1 -9816.413,E2 -9816.413} C_VEL
LIN {X 0,Y 424.581,Z 460.461,A -85,B 0,C 180,E1 -9817.611,E2 -9817.611} C_VEL
LIN {X 0,Y 424.82,Z 455.182,A -85,B 0,C 180,E1 -9818.564,E2 -9818.564} C_VEL
LIN {X 0,Y 425.145,Z 448.844,A -85,B 0,C 180,E1 -9819.516,E2 -9819.516} C_VEL
LIN {X 0,Y 425.645,Z 440.129,A -85,B 0,C 180,E1 -9820.586,E2 -9820.586} C_VEL
LIN {X 0,Y 426.195,Z 430.125,A -85,B 0,C 180,E1 -9821.535,E2 -9821.535} C_VEL
LIN {X 0,Y 426.602,Z 422.293,A -85,B 0,C 180,E1 -9822.126,E2 -9822.126} C_VEL
LIN {X 0,Y 426.192,Z 412.889,A -85,B 0,C 180,E1 -9822.707,E2 -9822.707} C_VEL
LIN {X 0,Y 425.319,Z 403.627,A -85,B 0,C 180,E1 -9823.155,E2 -9823.155} C_VEL
LIN {X 0,Y 424.343,Z 395.822,A -85,B 0,C 180,E1 -9823.469,E2 -9823.469} C_VEL
LIN {X 0,Y 424.632,Z 387.324,A -85,B 0,C 180,E1 -9826.837,E2 -9826.837} C_VEL
LIN {X 0,Y 424.908,Z 378.72,A -85,B 0,C 180,E1 -9830.326,E2 -9830.326} C_VEL
LIN {X 0,Y 425.284,Z 370.158,A -85,B 0,C 180,E1 -9833.884,E2 -9833.884} C_VEL
LIN {X 0,Y 425.722,Z 363.087,A -85,B 0,C 180,E1 -9836.943,E2 -9836.943} C_VEL
LIN {X 0,Y 426.416,Z 354.699,A -85,B 0,C 180,E1 -9840.727,E2 -9840.727} C_VEL
LIN {X 0,Y 426.733,Z 350.046,A -85,B 0,C 180,E1 -9842.922,E2 -9842.922} C_VEL
LIN {X 0,Y 426.445,Z 346.911,A -85,B 0,C 180,E1 -9844.51,E2 -9844.51} C_VEL
LIN {X 0,Y 425.335,Z 340.319,A -85,B 0,C 180,E1 -9848.102,E2 -9848.102} C_VEL
LIN {X 0,Y 425.281,Z 340.331,A -85,B 0,C 180,E1 -9851.379,E2 -9851.379} C_VEL
LIN {X 0,Y 425.292,Z 340.327,A -85,B 0,C 180,E1 -9854.717,E2 -9854.717} C_VEL
LIN {X 0,Y 425.296,Z 340.323,A -85,B 0,C 180,E1 -9858.042,E2 -9858.042} C_VEL
LIN {X 0,Y 425.299,Z 340.323,A -85,B 0,C 180,E1 -9861.101,E2 -9861.101} C_VEL
LIN {X 0,Y 425.305,Z 340.322,A -85,B 0,C 180,E1 -9864.664,E2 -9864.664} C_VEL
LIN {X 0,Y 425.271,Z 340.327,A -85,B 0,C 180,E1 -9868.073,E2 -9868.073} C_VEL
LIN {X 0,Y 425.338,Z 340.316,A -85,B 0,C 180,E1 -9871.368,E2 -9871.368} C_VEL
LIN {X 0,Y 425.3,Z 340.322,A -85,B 0,C 180,E1 -9874.554,E2 -9874.554} C_VEL
LIN {X 0,Y 425.295,Z 340.324,A -85,B 0,C 180,E1 -9877.661,E2 -9877.661} C_VEL
LIN {X 0,Y 425.368,Z 340.313,A -85,B 0,C 180,E1 -9880.704,E2 -9880.704} C_VEL
LIN {X 0,Y 425.395,Z 340.311,A -85,B 0,C 180,E1 -9883.688,E2 -9883.688} C_VEL
LIN {X 0,Y 425.419,Z 340.306,A -85,B 0,C 180,E1 -9887.598,E2 -9887.598} C_VEL
LIN {X 0,Y 425.414,Z 340.308,A -85,B 0,C 180,E1 -9891.449,E2 -9891.449} C_VEL
LIN {X 0,Y 425.546,Z 340.292,A -85,B 0,C 180,E1 -9894.312,E2 -9894.312} C_VEL
LIN {X 0,Y 425.577,Z 340.286,A -85,B 0,C 180,E1 -9898.106,E2 -9898.106} C_VEL
LIN {X 0,Y 425.707,Z 340.273,A -85,B 0,C 180,E1 -9899.999,E2 -9899.999} C_VEL
LIN {X 0,Y 425.549,Z 340.29,A -85,B 0,C 180,E1 -9902.839,E2 -9902.839} C_VEL
LIN {X 0,Y 425.554,Z 340.29,A -85,B 0,C 180,E1 -9905.686,E2 -9905.686} C_VEL
LIN {X 0,Y 425.412,Z 340.308,A -85,B 0,C 180,E1 -9908.55,E2 -9908.55} C_VEL
LIN {X 0,Y 425.416,Z 340.308,A -85,B 0,C 180,E1 -9912.401,E2 -9912.401} C_VEL
LIN {X 0,Y 425.348,Z 340.321,A -85,B 0,C 180,E1 -9915.328,E2 -9915.328} C_VEL
LIN {X 0,Y 425.232,Z 340.333,A -85,B 0,C 180,E1 -9917.306,E2 -9917.306} C_VEL
LIN {X 0,Y 424.985,Z 340.364,A -85,B 0,C 180,E1 -9919.503,E2 -9919.503} C_VEL
LIN {X 0,Y 424.823,Z 344.69,A -85,B 0,C 180,E1 -9923.392,E2 -9923.392} C_VEL
LIN {X 0,Y 424.633,Z 348.488,A -85,B 0,C 180,E1 -9926.651,E2 -9926.651} C_VEL
LIN {X 0,Y 424.544,Z 352.166,A -85,B 0,C 180,E1 -9929.776,E2 -9929.776} C_VEL
LIN {X 0,Y 424.398,Z 356.171,A -85,B 0,C 180,E1 -9933.124,E2 -9933.124} C_VEL
LIN {X 0,Y 424.323,Z 360.556,A -85,B 0,C 180,E1 -9936.668,E2 -9936.668} C_VEL
LIN {X 0,Y 426.429,Z 370.985,A -85,B 0,C 180,E1 -9937.166,E2 -9937.166} C_VEL
LIN {X 0,Y 427.364,Z 376.385,A -85,B 0,C 180,E1 -9937.477,E2 -9937.477} C_VEL
LIN {X 0,Y 426.944,Z 387.459,A -85,B 0,C 180,E1 -9938.21,E2 -9938.21} C_VEL
LIN {X 0,Y 426.513,Z 396.365,A -85,B 0,C 180,E1 -9938.979,E2 -9938.979} C_VEL
LIN {X 0,Y 426.152,Z 402.299,A -85,B 0,C 180,E1 -9939.593,E2 -9939.593} C_VEL
LIN {X 0,Y 425.852,Z 408.271,A -85,B 0,C 180,E1 -9940.319,E2 -9940.319} C_VEL
LIN {X 0,Y 425.461,Z 415.262,A -85,B 0,C 180,E1 -9941.355,E2 -9941.355} C_VEL
LIN {X 0,Y 425.164,Z 420.432,A -85,B 0,C 180,E1 -9942.276,E2 -9942.276} C_VEL
LIN {X 0,Y 424.813,Z 425.138,A -85,B 0,C 180,E1 -9943.286,E2 -9943.286} C_VEL
LIN {X 0,Y 424.706,Z 428.072,A -85,B 0,C 180,E1 -9944.026,E2 -9944.026} C_VEL
LIN {X 0,Y 424.435,Z 432.33,A -85,B 0,C 180,E1 -9945.397,E2 -9945.397} C_VEL
LIN {X 0,Y 424.186,Z 436.071,A -85,B 0,C 180,E1 -9947.21,E2 -9947.21} C_VEL
LIN {X 0,Y 424.115,Z 437.572,A -85,B 0,C 180,E1 -9948.482,E2 -9948.482} C_VEL
LIN {X 0,Y 424.033,Z 438.164,A -85,B 0,C 180,E1 -9949.729,E2 -9949.729} C_VEL
LIN {X 0,Y 424.045,Z 437.815,A -85,B 0,C 180,E1 -9951.164,E2 -9951.164} C_VEL
LIN {X 0,Y 424.148,Z 436.102,A -85,B 0,C 180,E1 -9952.685,E2 -9952.685} C_VEL
LIN {X 0,Y 424.277,Z 434.882,A -85,B 0,C 180,E1 -9953.392,E2 -9953.392} C_VEL
LIN {X 0,Y 424.383,Z 432.148,A -85,B 0,C 180,E1 -9954.575,E2 -9954.575} C_VEL
LIN {X 0,Y 424.614,Z 427.142,A -85,B 0,C 180,E1 -9956.121,E2 -9956.121} C_VEL
LIN {X 0,Y 424.872,Z 422.347,A -85,B 0,C 180,E1 -9957.244,E2 -9957.244} C_VEL
LIN {X 0,Y 425.216,Z 416.5,A -85,B 0,C 180,E1 -9958.347,E2 -9958.347} C_VEL
LIN {X 0,Y 425.571,Z 410.032,A -85,B 0,C 180,E1 -9959.343,E2 -9959.343} C_VEL
LIN {X 0,Y 425.872,Z 403.422,A -85,B 0,C 180,E1 -9960.188,E2 -9960.188} C_VEL
LIN {X 0,Y 426.332,Z 395.098,A -85,B 0,C 180,E1 -9961.06,E2 -9961.06} C_VEL
LIN {X 0,Y 426.746,Z 384.483,A -85,B 0,C 180,E1 -9961.939,E2 -9961.939} C_VEL
LIN {X 0,Y 427.087,Z 375.497,A -85,B 0,C 180,E1 -9962.496,E2 -9962.496} C_VEL
LIN {X 0,Y 425.259,Z 364.813,A -85,B 0,C 180,E1 -9963.046,E2 -9963.046} C_VEL
LIN {X 0,Y 424.327,Z 359.761,A -85,B 0,C 180,E1 -9963.275,E2 -9963.275} C_VEL
LIN {X 0,Y 424.311,Z 355.583,A -85,B 0,C 180,E1 -9966.576,E2 -9966.576} C_VEL
LIN {X 0,Y 424.388,Z 351.735,A -85,B 0,C 180,E1 -9969.648,E2 -9969.648} C_VEL
LIN {X 0,Y 424.522,Z 348.028,A -85,B 0,C 180,E1 -9972.662,E2 -9972.662} C_VEL
LIN {X 0,Y 424.61,Z 344.413,A -85,B 0,C 180,E1 -9975.623,E2 -9975.623} C_VEL
LIN {X 0,Y 424.781,Z 340.909,A -85,B 0,C 180,E1 -9978.547,E2 -9978.547} C_VEL
LIN {X 0,Y 424.871,Z 340.376,A -85,B 0,C 180,E1 -9979.515,E2 -9979.515} C_VEL
LIN {X 0,Y 425.401,Z 340.311,A -85,B 0,C 180,E1 -9982.404,E2 -9982.404} C_VEL
LIN {X 0,Y 425.478,Z 340.298,A -85,B 0,C 180,E1 -9984.554,E2 -9984.554} C_VEL
LIN {X 0,Y 425.565,Z 340.289,A -85,B 0,C 180,E1 -9988.106,E2 -9988.106} C_VEL
LIN {X 0,Y 425.538,Z 340.289,A -85,B 0,C 180,E1 -9988.699,E2 -9988.699} C_VEL
LIN {X 0,Y 424.871,Z 340.375,A -85,B 0,C 180,E1 -9989.489,E2 -9989.489} C_VEL
LIN {X 0,Y 422.009,Z 340.73,A -85,B 0,C 180,E1 -9990.772,E2 -9990.772} C_VEL
LIN {X 0,Y 419.597,Z 341.032,A -85,B 0,C 180,E1 -9991.808,E2 -9991.808} C_VEL
LIN {X 0,Y 418.576,Z 341.159,A -85,B 0,C 180,E1 -9992.609,E2 -9992.609} C_VEL
LIN {X 0,Y 418.502,Z 341.167,A -85,B 0,C 180,E1 -9992.88,E2 -9992.88} C_VEL
LIN {X 0,Y 418.523,Z 341.167,A -85,B 0,C 180,E1 -9995.781,E2 -9995.781} C_VEL
LIN {X 0,Y 418.389,Z 341.18,A -85,B 0,C 180,E1 -9998.694,E2 -9998.694} C_VEL
LIN {X 0,Y 418.321,Z 341.192,A -85,B 0,C 180,E1 -10001.63,E2 -10001.63} C_VEL
LIN {X 0,Y 418.293,Z 341.192,A -85,B 0,C 180,E1 -10004.596,E2 -10004.596} C_VEL
LIN {X 0,Y 418.275,Z 341.198,A -85,B 0,C 180,E1 -10007.603,E2 -10007.603} C_VEL
LIN {X 0,Y 418.237,Z 341.199,A -85,B 0,C 180,E1 -10010.662,E2 -10010.662} C_VEL
LIN {X 0,Y 418.274,Z 341.198,A -85,B 0,C 180,E1 -10013.78,E2 -10013.78} C_VEL
LIN {X 0,Y 418.296,Z 341.194,A -85,B 0,C 180,E1 -10017.07,E2 -10017.07} C_VEL
LIN {X 0,Y 418.246,Z 341.198,A -85,B 0,C 180,E1 -10020.27,E2 -10020.27} C_VEL
LIN {X 0,Y 418.234,Z 341.202,A -85,B 0,C 180,E1 -10023.677,E2 -10023.677} C_VEL
LIN {X 0,Y 418.233,Z 341.204,A -85,B 0,C 180,E1 -10027.223,E2 -10027.223} C_VEL
LIN {X 0,Y 418.252,Z 341.199,A -85,B 0,C 180,E1 -10029.68,E2 -10029.68} C_VEL
LIN {X 0,Y 418.27,Z 341.196,A -85,B 0,C 180,E1 -10032.329,E2 -10032.329} C_VEL
LIN {X 0,Y 418.259,Z 341.199,A -85,B 0,C 180,E1 -10035.114,E2 -10035.114} C_VEL
LIN {X 0,Y 418.277,Z 341.195,A -85,B 0,C 180,E1 -10037.773,E2 -10037.773} C_VEL
LIN {X 0,Y 418.252,Z 341.199,A -85,B 0,C 180,E1 -10041.56,E2 -10041.56} C_VEL
LIN {X 0,Y 418.245,Z 341.201,A -85,B 0,C 180,E1 -10045.159,E2 -10045.159} C_VEL
LIN {X 0,Y 418.234,Z 341.2,A -85,B 0,C 180,E1 -10047.472,E2 -10047.472} C_VEL
LIN {X 0,Y 418.262,Z 341.199,A -85,B 0,C 180,E1 -10050.894,E2 -10050.894} C_VEL
LIN {X 0,Y 418.257,Z 341.199,A -85,B 0,C 180,E1 -10054.096,E2 -10054.096} C_VEL
LIN {X 0,Y 418.281,Z 341.194,A -85,B 0,C 180,E1 -10057.531,E2 -10057.531} C_VEL
LIN {X 0,Y 418.303,Z 341.194,A -85,B 0,C 180,E1 -10060.366,E2 -10060.366} C_VEL
LIN {X 0,Y 418.312,Z 341.19,A -85,B 0,C 180,E1 -10063.406,E2 -10063.406} C_VEL
LIN {X 0,Y 418.342,Z 341.187,A -85,B 0,C 180,E1 -10066.995,E2 -10066.995} C_VEL
LIN {X 0,Y 418.347,Z 341.188,A -85,B 0,C 180,E1 -10070.33,E2 -10070.33} C_VEL
LIN {X 0,Y 418.482,Z 341.169,A -85,B 0,C 180,E1 -10073.25,E2 -10073.25} C_VEL
LIN {X 0,Y 418.33,Z 341.187,A -85,B 0,C 180,E1 -10075.182,E2 -10075.182} C_VEL
LIN {X 0,Y 418.533,Z 341.166,A -85,B 0,C 180,E1 -10078.076,E2 -10078.076} C_VEL
LIN {X 0,Y 418.661,Z 341.149,A -85,B 0,C 180,E1 -10080.001,E2 -10080.001} C_VEL
LIN {X 0,Y 418.502,Z 341.166,A -85,B 0,C 180,E1 -10082.889,E2 -10082.889} C_VEL
LIN {X 0,Y 418.483,Z 341.169,A -85,B 0,C 180,E1 -10086.752,E2 -10086.752} C_VEL
LIN {X 0,Y 418.35,Z 341.188,A -85,B 0,C 180,E1 -10089.672,E2 -10089.672} C_VEL
LIN {X 0,Y 418.345,Z 341.187,A -85,B 0,C 180,E1 -10093.007,E2 -10093.007} C_VEL
LIN {X 0,Y 418.303,Z 341.192,A -85,B 0,C 180,E1 -10096.737,E2 -10096.737} C_VEL
LIN {X 0,Y 418.261,Z 341.2,A -85,B 0,C 180,E1 -10099.792,E2 -10099.792} C_VEL
LIN {X 0,Y 418.229,Z 341.201,A -85,B 0,C 180,E1 -10102.737,E2 -10102.737} C_VEL
LIN {X 0,Y 418.263,Z 341.198,A -85,B 0,C 180,E1 -10105.905,E2 -10105.905} C_VEL
LIN {X 0,Y 418.267,Z 341.198,A -85,B 0,C 180,E1 -10109.162,E2 -10109.162} C_VEL
LIN {X 0,Y 418.25,Z 341.2,A -85,B 0,C 180,E1 -10112.845,E2 -10112.845} C_VEL
LIN {X 0,Y 418.242,Z 341.199,A -85,B 0,C 180,E1 -10116.24,E2 -10116.24} C_VEL
LIN {X 0,Y 418.246,Z 341.198,A -85,B 0,C 180,E1 -10119.683,E2 -10119.683} C_VEL
LIN {X 0,Y 418.226,Z 341.202,A -85,B 0,C 180,E1 -10122.323,E2 -10122.323} C_VEL
LIN {X 0,Y 418.236,Z 341.202,A -85,B 0,C 180,E1 -10125.111,E2 -10125.111} C_VEL
LIN {X 0,Y 418.237,Z 341.199,A -85,B 0,C 180,E1 -10127.769,E2 -10127.769} C_VEL
LIN {X 0,Y 418.255,Z 341.199,A -85,B 0,C 180,E1 -10130.62,E2 -10130.62} C_VEL
LIN {X 0,Y 418.286,Z 341.293,A -85,B 0,C 180,E1 -10132.364,E2 -10132.364} C_VEL
LIN {X 0,Y 419.31,Z 347.019,A -85,B 0,C 180,E1 -10135.261,E2 -10135.261} C_VEL
LIN {X 0,Y 419.663,Z 350.33,A -85,B 0,C 180,E1 -10136.861,E2 -10136.861} C_VEL
LIN {X 0,Y 419.308,Z 355.555,A -85,B 0,C 180,E1 -10139.265,E2 -10139.265} C_VEL
LIN {X 0,Y 418.865,Z 361.637,A -85,B 0,C 180,E1 -10141.98,E2 -10141.98} C_VEL
LIN {X 0,Y 418.374,Z 368.968,A -85,B 0,C 180,E1 -10145.17,E2 -10145.17} C_VEL
LIN {X 0,Y 417.928,Z 377.535,A -85,B 0,C 180,E1 -10148.806,E2 -10148.806} C_VEL
LIN {X 0,Y 417.593,Z 386.129,A -85,B 0,C 180,E1 -10152.367,E2 -10152.367} C_VEL
LIN {X 0,Y 417.297,Z 394.704,A -85,B 0,C 180,E1 -10155.867,E2 -10155.867} C_VEL
LIN {X 0,Y 417.272,Z 396.25,A -85,B 0,C 180,E1 -10156.492,E2 -10156.492} C_VEL
LIN {X 0,Y 418.683,Z 408.911,A -85,B 0,C 180,E1 -10157.008,E2 -10157.008} C_VEL
LIN {X 0,Y 419.416,Z 418.297,A -85,B 0,C 180,E1 -10157.542,E2 -10157.542} C_VEL
LIN {X 0,Y 419.224,Z 426.95,A -85,B 0,C 180,E1 -10158.151,E2 -10158.151} C_VEL
LIN {X 0,Y 418.747,Z 435.23,A -85,B 0,C 180,E1 -10158.873,E2 -10158.873} C_VEL
LIN {X 0,Y 418.37,Z 443.094,A -85,B 0,C 180,E1 -10159.72,E2 -10159.72} C_VEL
LIN {X 0,Y 417.99,Z 449.599,A -85,B 0,C 180,E1 -10160.566,E2 -10160.566} C_VEL
LIN {X 0,Y 417.695,Z 455.801,A -85,B 0,C 180,E1 -10161.535,E2 -10161.535} C_VEL
LIN {X 0,Y 417.458,Z 460.949,A -85,B 0,C 180,E1 -10162.504,E2 -10162.504} C_VEL
LIN {X 0,Y 417.194,Z 466.033,A -85,B 0,C 180,E1 -10163.675,E2 -10163.675} C_VEL
LIN {X 0,Y 417.164,Z 471.07,A -85,B 0,C 180,E1 -10165.169,E2 -10165.169} C_VEL
LIN {X 0,Y 417.058,Z 473.435,A -85,B 0,C 180,E1 -10166.136,E2 -10166.136} C_VEL
LIN {X 0,Y 417.105,Z 475.252,A -85,B 0,C 180,E1 -10167.104,E2 -10167.104} C_VEL
LIN {X 0,Y 417.094,Z 476.558,A -85,B 0,C 180,E1 -10168.07,E2 -10168.07} C_VEL
LIN {X 0,Y 417.054,Z 477.378,A -85,B 0,C 180,E1 -10169.036,E2 -10169.036} C_VEL
LIN {X 0,Y 417.051,Z 477.674,A -85,B 0,C 180,E1 -10170.001,E2 -10170.001} C_VEL
LIN {X 0,Y 417.055,Z 477.384,A -85,B 0,C 180,E1 -10170.967,E2 -10170.967} C_VEL
LIN {X 0,Y 417.093,Z 476.62,A -85,B 0,C 180,E1 -10171.932,E2 -10171.932} C_VEL
LIN {X 0,Y 417.09,Z 475.374,A -85,B 0,C 180,E1 -10172.899,E2 -10172.899} C_VEL
LIN {X 0,Y 417.092,Z 472.446,A -85,B 0,C 180,E1 -10174.35,E2 -10174.35} C_VEL
LIN {X 0,Y 417.178,Z 469.796,A -85,B 0,C 180,E1 -10175.318,E2 -10175.318} C_VEL
LIN {X 0,Y 417.235,Z 466.165,A -85,B 0,C 180,E1 -10176.377,E2 -10176.377} C_VEL
LIN {X 0,Y 417.483,Z 461.368,A -85,B 0,C 180,E1 -10177.498,E2 -10177.498} C_VEL
LIN {X 0,Y 417.701,Z 456.342,A -85,B 0,C 180,E1 -10178.467,E2 -10178.467} C_VEL
LIN {X 0,Y 418.034,Z 450.3,A -85,B 0,C 180,E1 -10179.435,E2 -10179.435} C_VEL
LIN {X 0,Y 418.459,Z 442.967,A -85,B 0,C 180,E1 -10180.403,E2 -10180.403} C_VEL
LIN {X 0,Y 418.879,Z 435.159,A -85,B 0,C 180,E1 -10181.249,E2 -10181.249} C_VEL
LIN {X 0,Y 419.358,Z 426.965,A -85,B 0,C 180,E1 -10181.971,E2 -10181.971} C_VEL
LIN {X 0,Y 419.662,Z 420.327,A -85,B 0,C 180,E1 -10182.453,E2 -10182.453} C_VEL
LIN {X 0,Y 419.171,Z 412.01,A -85,B 0,C 180,E1 -10182.969,E2 -10182.969} C_VEL
LIN {X 0,Y 418.288,Z 403.15,A -85,B 0,C 180,E1 -10183.406,E2 -10183.406} C_VEL
LIN {X 0,Y 417.251,Z 395.512,A -85,B 0,C 180,E1 -10183.703,E2 -10183.703} C_VEL
LIN {X 0,Y 417.514,Z 388.295,A -85,B 0,C 180,E1 -10186.629,E2 -10186.629} C_VEL
LIN {X 0,Y 417.806,Z 379.702,A -85,B 0,C 180,E1 -10190.173,E2 -10190.173} C_VEL
LIN {X 0,Y 418.202,Z 371.205,A -85,B 0,C 180,E1 -10193.787,E2 -10193.787} C_VEL
LIN {X 0,Y 418.693,Z 363.985,A -85,B 0,C 180,E1 -10196.951,E2 -10196.951} C_VEL
LIN {X 0,Y 419.41,Z 355.781,A -85,B 0,C 180,E1 -10200.737,E2 -10200.737} C_VEL
LIN {X 0,Y 419.736,Z 350.796,A -85,B 0,C 180,E1 -10203.154,E2 -10203.154} C_VEL
LIN {X 0,Y 419.185,Z 346.617,A -85,B 0,C 180,E1 -10205.34,E2 -10205.34} C_VEL
LIN {X 0,Y 418.282,Z 341.199,A -85,B 0,C 180,E1 -10208.44,E2 -10208.44} C_VEL
LIN {X 0,Y 418.247,Z 341.207,A -85,B 0,C 180,E1 -10212.234,E2 -10212.234} C_VEL
LIN {X 0,Y 418.243,Z 341.206,A -85,B 0,C 180,E1 -10215.109,E2 -10215.109} C_VEL
LIN {X 0,Y 418.246,Z 341.202,A -85,B 0,C 180,E1 -10217.767,E2 -10217.767} C_VEL
LIN {X 0,Y 418.249,Z 341.2,A -85,B 0,C 180,E1 -10220.621,E2 -10220.621} C_VEL
LIN {X 0,Y 418.249,Z 341.2,A -85,B 0,C 180,E1 -10223.976,E2 -10223.976} C_VEL
LIN {X 0,Y 418.264,Z 341.199,A -85,B 0,C 180,E1 -10227.156,E2 -10227.156} C_VEL
LIN {X 0,Y 418.276,Z 341.196,A -85,B 0,C 180,E1 -10230.895,E2 -10230.895} C_VEL
LIN {X 0,Y 418.277,Z 341.198,A -85,B 0,C 180,E1 -10234.096,E2 -10234.096} C_VEL
LIN {X 0,Y 418.246,Z 341.2,A -85,B 0,C 180,E1 -10237.264,E2 -10237.264} C_VEL
LIN {X 0,Y 418.29,Z 341.195,A -85,B 0,C 180,E1 -10240.364,E2 -10240.364} C_VEL
LIN {X 0,Y 418.324,Z 341.191,A -85,B 0,C 180,E1 -10243.404,E2 -10243.404} C_VEL
LIN {X 0,Y 418.353,Z 341.189,A -85,B 0,C 180,E1 -10246.999,E2 -10246.999} C_VEL
LIN {X 0,Y 418.345,Z 341.189,A -85,B 0,C 180,E1 -10250.328,E2 -10250.328} C_VEL
LIN {X 0,Y 418.465,Z 341.173,A -85,B 0,C 180,E1 -10253.248,E2 -10253.248} C_VEL
LIN {X 0,Y 418.337,Z 341.19,A -85,B 0,C 180,E1 -10255.181,E2 -10255.181} C_VEL
LIN {X 0,Y 418.546,Z 341.161,A -85,B 0,C 180,E1 -10258.075,E2 -10258.075} C_VEL
LIN {X 0,Y 418.676,Z 341.149,A -85,B 0,C 180,E1 -10259.999,E2 -10259.999} C_VEL
LIN {X 0,Y 418.504,Z 341.167,A -85,B 0,C 180,E1 -10262.887,E2 -10262.887} C_VEL
LIN {X 0,Y 418.475,Z 341.172,A -85,B 0,C 180,E1 -10266.626,E2 -10266.626} C_VEL
LIN {X 0,Y 418.343,Z 341.19,A -85,B 0,C 180,E1 -10269.67,E2 -10269.67} C_VEL
LIN {X 0,Y 418.35,Z 341.19,A -85,B 0,C 180,E1 -10272.999,E2 -10272.999} C_VEL
LIN {X 0,Y 418.309,Z 341.198,A -85,B 0,C 180,E1 -10276.595,E2 -10276.595} C_VEL
LIN {X 0,Y 417.917,Z 341.424,A -85,B 0,C 180,E1 -10279.652,E2 -10279.652} C_VEL
LIN {X 0,Y 417.765,Z 344.894,A -85,B 0,C 180,E1 -10282.762,E2 -10282.762} C_VEL
LIN {X 0,Y 417.62,Z 348.459,A -85,B 0,C 180,E1 -10285.946,E2 -10285.946} C_VEL
LIN {X 0,Y 417.496,Z 352.268,A -85,B 0,C 180,E1 -10289.219,E2 -10289.219} C_VEL
LIN {X 0,Y 417.369,Z 356.303,A -85,B 0,C 180,E1 -10292.653,E2 -10292.653} C_VEL
LIN {X 0,Y 417.238,Z 360.482,A -85,B 0,C 180,E1 -10296.123,E2 -10296.123} C_VEL
LIN {X 0,Y 417.276,Z 360.965,A -85,B 0,C 180,E1 -10296.418,E2 -10296.418} C_VEL
LIN {X 0,Y 419.467,Z 371.658,A -85,B 0,C 180,E1 -10296.945,E2 -10296.945} C_VEL
LIN {X 0,Y 420.459,Z 378.748,A -85,B 0,C 180,E1 -10297.369,E2 -10297.369} C_VEL
LIN {X 0,Y 420.018,Z 388.474,A -85,B 0,C 180,E1 -10298.049,E2 -10298.049} C_VEL
LIN {X 0,Y 419.591,Z 396.501,A -85,B 0,C 180,E1 -10298.755,E2 -10298.755} C_VEL
LIN {X 0,Y 419.133,Z 404.144,A -85,B 0,C 180,E1 -10299.58,E2 -10299.58} C_VEL
LIN {X 0,Y 418.684,Z 411.648,A -85,B 0,C 180,E1 -10300.574,E2 -10300.574} C_VEL
LIN {X 0,Y 418.359,Z 417.782,A -85,B 0,C 180,E1 -10301.569,E2 -10301.569} C_VEL
LIN {X 0,Y 417.838,Z 424.749,A -85,B 0,C 180,E1 -10302.973,E2 -10302.973} C_VEL
LIN {X 0,Y 417.546,Z 429.769,A -85,B 0,C 180,E1 -10304.327,E2 -10304.327} C_VEL
LIN {X 0,Y 417.335,Z 433.52,A -85,B 0,C 180,E1 -10305.668,E2 -10305.668} C_VEL
LIN {X 0,Y 417.222,Z 435.19,A -85,B 0,C 180,E1 -10306.411,E2 -10306.411} C_VEL
LIN {X 0,Y 417.042,Z 437.342,A -85,B 0,C 180,E1 -10307.856,E2 -10307.856} C_VEL
LIN {X 0,Y 416.951,Z 438.382,A -85,B 0,C 180,E1 -10309.33,E2 -10309.33} C_VEL
LIN {X 0,Y 416.947,Z 438.277,A -85,B 0,C 180,E1 -10310.836,E2 -10310.836} C_VEL
LIN {X 0,Y 417.033,Z 436.953,A -85,B 0,C 180,E1 -10312.376,E2 -10312.376} C_VEL
LIN {X 0,Y 417.244,Z 434.132,A -85,B 0,C 180,E1 -10313.948,E2 -10313.948} C_VEL
LIN {X 0,Y 417.428,Z 429.633,A -85,B 0,C 180,E1 -10315.584,E2 -10315.584} C_VEL
LIN {X 0,Y 417.694,Z 425.138,A -85,B 0,C 180,E1 -10316.795,E2 -10316.795} C_VEL
LIN {X 0,Y 418.134,Z 417.747,A -85,B 0,C 180,E1 -10318.314,E2 -10318.314} C_VEL
LIN {X 0,Y 418.473,Z 412.231,A -85,B 0,C 180,E1 -10319.217,E2 -10319.217} C_VEL
LIN {X 0,Y 418.87,Z 404.342,A -85,B 0,C 180,E1 -10320.271,E2 -10320.271} C_VEL
LIN {X 0,Y 419.227,Z 397.269,A -85,B 0,C 180,E1 -10321.048,E2 -10321.048} C_VEL
LIN {X 0,Y 419.638,Z 389.351,A -85,B 0,C 180,E1 -10321.762,E2 -10321.762} C_VEL
LIN {X 0,Y 420.015,Z 380.666,A -85,B 0,C 180,E1 -10322.391,E2 -10322.391} C_VEL
LIN {X 0,Y 420.136,Z 376.431,A -85,B 0,C 180,E1 -10322.657,E2 -10322.657} C_VEL
LIN {X 0,Y 418.263,Z 365.504,A -85,B 0,C 180,E1 -10323.237,E2 -10323.237} C_VEL
LIN {X 0,Y 417.233,Z 360.072,A -85,B 0,C 180,E1 -10323.48,E2 -10323.48} C_VEL
LIN {X 0,Y 417.248,Z 356.705,A -85,B 0,C 180,E1 -10326.155,E2 -10326.155} C_VEL
LIN {X 0,Y 417.305,Z 352.827,A -85,B 0,C 180,E1 -10329.287,E2 -10329.287} C_VEL
LIN {X 0,Y 417.45,Z 349.058,A -85,B 0,C 180,E1 -10332.359,E2 -10332.359} C_VEL
LIN {X 0,Y 417.55,Z 345.429,A -85,B 0,C 180,E1 -10335.375,E2 -10335.375} C_VEL
LIN {X 0,Y 417.724,Z 341.897,A -85,B 0,C 180,E1 -10338.351,E2 -10338.351} C_VEL
LIN {X 0,Y 417.787,Z 341.258,A -85,B 0,C 180,E1 -10339.335,E2 -10339.335} C_VEL
LIN {X 0,Y 418.355,Z 341.189,A -85,B 0,C 180,E1 -10342.359,E2 -10342.359} C_VEL
LIN {X 0,Y 418.49,Z 341.171,A -85,B 0,C 180,E1 -10344.216,E2 -10344.216} C_VEL
LIN {X 0,Y 418.535,Z 341.165,A -85,B 0,C 180,E1 -10348.074,E2 -10348.074} C_VEL
LIN {X 0,Y 418.662,Z 341.15,A -85,B 0,C 180,E1 -10349.999,E2 -10349.999} C_VEL
LIN {X 0,Y 418.502,Z 341.167,A -85,B 0,C 180,E1 -10352.88,E2 -10352.88} C_VEL
LIN {X 0,Y 417.854,Z 341.25,A -85,B 0,C 180,E1 -10353.683,E2 -10353.683} C_VEL
LIN {X 0,Y 415,Z 341.606,A -85,B 0,C 180,E1 -10354.987,E2 -10354.987} C_VEL
LIN {X 0,Y 412.571,Z 341.908,A -85,B 0,C 180,E1 -10356.04,E2 -10356.04} C_VEL
LIN {X 0,Y 411.528,Z 342.035,A -85,B 0,C 180,E1 -10356.854,E2 -10356.854} C_VEL
LIN {X 0,Y 411.444,Z 342.045,A -85,B 0,C 180,E1 -10357.13,E2 -10357.13} C_VEL
LIN {X 0,Y 411.286,Z 342.065,A -85,B 0,C 180,E1 -10360.833,E2 -10360.833} C_VEL
LIN {X 0,Y 411.252,Z 342.073,A -85,B 0,C 180,E1 -10363.841,E2 -10363.841} C_VEL
LIN {X 0,Y 411.244,Z 342.071,A -85,B 0,C 180,E1 -10366.888,E2 -10366.888} C_VEL
LIN {X 0,Y 411.217,Z 342.077,A -85,B 0,C 180,E1 -10369.986,E2 -10369.986} C_VEL
LIN {X 0,Y 411.189,Z 342.08,A -85,B 0,C 180,E1 -10373.147,E2 -10373.147} C_VEL
LIN {X 0,Y 411.224,Z 342.073,A -85,B 0,C 180,E1 -10376.38,E2 -10376.38} C_VEL
LIN {X 0,Y 411.197,Z 342.079,A -85,B 0,C 180,E1 -10379.711,E2 -10379.711} C_VEL
LIN {X 0,Y 411.192,Z 342.08,A -85,B 0,C 180,E1 -10383.155,E2 -10383.155} C_VEL
LIN {X 0,Y 411.181,Z 342.079,A -85,B 0,C 180,E1 -10386.553,E2 -10386.553} C_VEL
LIN {X 0,Y 411.214,Z 342.075,A -85,B 0,C 180,E1 -10389.73,E2 -10389.73} C_VEL
LIN {X 0,Y 411.213,Z 342.078,A -85,B 0,C 180,E1 -10393.126,E2 -10393.126} C_VEL
LIN {X 0,Y 411.216,Z 342.074,A -85,B 0,C 180,E1 -10395.872,E2 -10395.872} C_VEL
LIN {X 0,Y 411.195,Z 342.079,A -85,B 0,C 180,E1 -10398.764,E2 -10398.764} C_VEL
LIN {X 0,Y 411.19,Z 342.077,A -85,B 0,C 180,E1 -10402.028,E2 -10402.028} C_VEL
LIN {X 0,Y 411.191,Z 342.077,A -85,B 0,C 180,E1 -10405.667,E2 -10405.667} C_VEL
LIN {X 0,Y 411.185,Z 342.079,A -85,B 0,C 180,E1 -10409.154,E2 -10409.154} C_VEL
LIN {X 0,Y 411.245,Z 342.073,A -85,B 0,C 180,E1 -10412.523,E2 -10412.523} C_VEL
LIN {X 0,Y 411.215,Z 342.074,A -85,B 0,C 180,E1 -10415.785,E2 -10415.785} C_VEL
LIN {X 0,Y 411.224,Z 342.074,A -85,B 0,C 180,E1 -10418.969,E2 -10418.969} C_VEL
LIN {X 0,Y 411.24,Z 342.073,A -85,B 0,C 180,E1 -10422.086,E2 -10422.086} C_VEL
LIN {X 0,Y 411.254,Z 342.069,A -85,B 0,C 180,E1 -10425.148,E2 -10425.148} C_VEL
LIN {X 0,Y 411.286,Z 342.068,A -85,B 0,C 180,E1 -10428.168,E2 -10428.168} C_VEL
LIN {X 0,Y 411.469,Z 342.046,A -85,B 0,C 180,E1 -10432.147,E2 -10432.147} C_VEL
LIN {X 0,Y 411.464,Z 342.046,A -85,B 0,C 180,E1 -10434.119,E2 -10434.119} C_VEL
LIN {X 0,Y 411.502,Z 342.042,A -85,B 0,C 180,E1 -10438.044,E2 -10438.044} C_VEL
LIN {X 0,Y 411.63,Z 342.025,A -85,B 0,C 180,E1 -10440.001,E2 -10440.001} C_VEL
LIN {X 0,Y 411.458,Z 342.044,A -85,B 0,C 180,E1 -10442.938,E2 -10442.938} C_VEL
LIN {X 0,Y 411.45,Z 342.045,A -85,B 0,C 180,E1 -10446.868,E2 -10446.868} C_VEL
LIN {X 0,Y 411.298,Z 342.067,A -85,B 0,C 180,E1 -10449.839,E2 -10449.839} C_VEL
LIN {X 0,Y 411.303,Z 342.065,A -85,B 0,C 180,E1 -10453.11,E2 -10453.11} C_VEL
LIN {X 0,Y 411.248,Z 342.071,A -85,B 0,C 180,E1 -10456.89,E2 -10456.89} C_VEL
LIN {X 0,Y 411.221,Z 342.075,A -85,B 0,C 180,E1 -10459.988,E2 -10459.988} C_VEL
LIN {X 0,Y 411.195,Z 342.079,A -85,B 0,C 180,E1 -10463.149,E2 -10463.149} C_VEL
